// TIA Portal V17 export
// export: Created 2022-06-27T14:00:09.5735646Z, ExportSetting WithDefaults, DisplayName Totally Integrated Automation Portal, DisplayVersion V17 Update 3, DisplayName TIA Portal Openness, DisplayVersion V17 Update 3, DisplayName TIA Portal Version Control Interface, DisplayVersion V17, DisplayName SINAMICS Startdrive Advanced, DisplayVersion V17 Update1, DisplayName SINAMICS Startdrive G110M, G120, G120C, G120D, G120P, G115D, DisplayVersion V17 Update1, DisplayName SINAMICS Startdrive G130, G150, S120, S150, SINAMICS MV, S210, DisplayVersion V17 Update1, DisplayName STEP 7 Professional, DisplayVersion V17 Update 3, DisplayName STEP 7 Safety, DisplayVersion V17, DisplayName WinCC UA Professional, DisplayVersion V17 Update 3
FUNCTION_BLOCK "S0822_RECIPE_FAILURES"   // FB822, LAD
{ S7_Optimized_Access := 'TRUE' }
VERSION : 0.1
// stored: AutoNumber false, IsIECCheckEnabled false, IsRetainMemResEnabled false, MemoryReserve 100, SetENOAutomatically false, UDAEnableTagReadback false
   VAR
      ls_wFaultRecipe : Word;
      ls_dwC1FaultProfile : DWord;
      ls_dwC2FaultProfile : DWord;
      ls_bRecipeOk : Bool;
   END_VAR
BEGIN

REGION Network 1: Falha Receita - Nome Receita
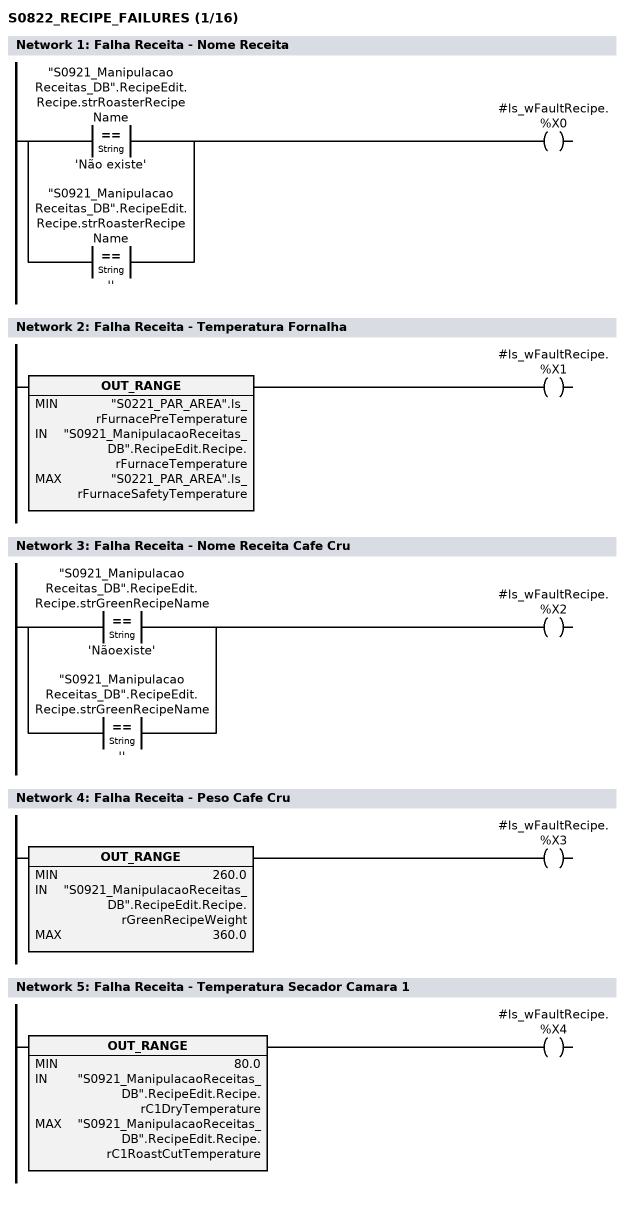
   RUNG wire#powerrail
      { S7_Templates := "SrcType := String" } EQ_Contact(in1 := "S0921_ManipulacaoReceitas_DB".RecipeEdit.Recipe.strRoasterRecipeName, in2 := 'Não existe')
      wire#w1
      Coil( #ls_wFaultRecipe.%X0 )
   END_RUNG
   RUNG wire#powerrail
      { S7_Templates := "SrcType := String" } EQ_Contact(in1 := "S0921_ManipulacaoReceitas_DB".RecipeEdit.Recipe.strRoasterRecipeName, in2 := '')
   END_RUNG wire#w1
   // the same network as SCL:
   #ls_wFaultRecipe.%X0 := ("S0921_ManipulacaoReceitas_DB".RecipeEdit.Recipe.strRoasterRecipeName = 'Não existe') OR ("S0921_ManipulacaoReceitas_DB".RecipeEdit.Recipe.strRoasterRecipeName = '');
END_REGION

REGION Network 2: Falha Receita - Temperatura Fornalha
   #ls_wFaultRecipe.%X1 := ("S0921_ManipulacaoReceitas_DB".RecipeEdit.Recipe.rFurnaceTemperature < "S0221_PAR_AREA".ls_rFurnacePreTemperature) OR ("S0921_ManipulacaoReceitas_DB".RecipeEdit.Recipe.rFurnaceTemperature > "S0221_PAR_AREA".ls_rFurnaceSafetyTemperature);
END_REGION

REGION Network 3: Falha Receita - Nome Receita Cafe Cru
   RUNG wire#powerrail
      { S7_Templates := "SrcType := String" } EQ_Contact(in1 := "S0921_ManipulacaoReceitas_DB".RecipeEdit.Recipe.strGreenRecipeName, in2 := 'Nãoexiste')
      wire#w1
      Coil( #ls_wFaultRecipe.%X2 )
   END_RUNG
   RUNG wire#powerrail
      { S7_Templates := "SrcType := String" } EQ_Contact(in1 := "S0921_ManipulacaoReceitas_DB".RecipeEdit.Recipe.strGreenRecipeName, in2 := '')
   END_RUNG wire#w1
   // the same network as SCL:
   #ls_wFaultRecipe.%X2 := ("S0921_ManipulacaoReceitas_DB".RecipeEdit.Recipe.strGreenRecipeName = 'Nãoexiste') OR ("S0921_ManipulacaoReceitas_DB".RecipeEdit.Recipe.strGreenRecipeName = '');
END_REGION

REGION Network 4: Falha Receita - Peso Cafe Cru
   #ls_wFaultRecipe.%X3 := ("S0921_ManipulacaoReceitas_DB".RecipeEdit.Recipe.rGreenRecipeWeight < 260.0) OR ("S0921_ManipulacaoReceitas_DB".RecipeEdit.Recipe.rGreenRecipeWeight > 360.0);
END_REGION

REGION Network 5: Falha Receita - Temperatura Secador Camara 1
   #ls_wFaultRecipe.%X4 := ("S0921_ManipulacaoReceitas_DB".RecipeEdit.Recipe.rC1DryTemperature < 80.0) OR ("S0921_ManipulacaoReceitas_DB".RecipeEdit.Recipe.rC1DryTemperature > "S0921_ManipulacaoReceitas_DB".RecipeEdit.Recipe.rC1RoastCutTemperature);
END_REGION

REGION Network 6: Falha Receita - Temperatura Secador Camara 2
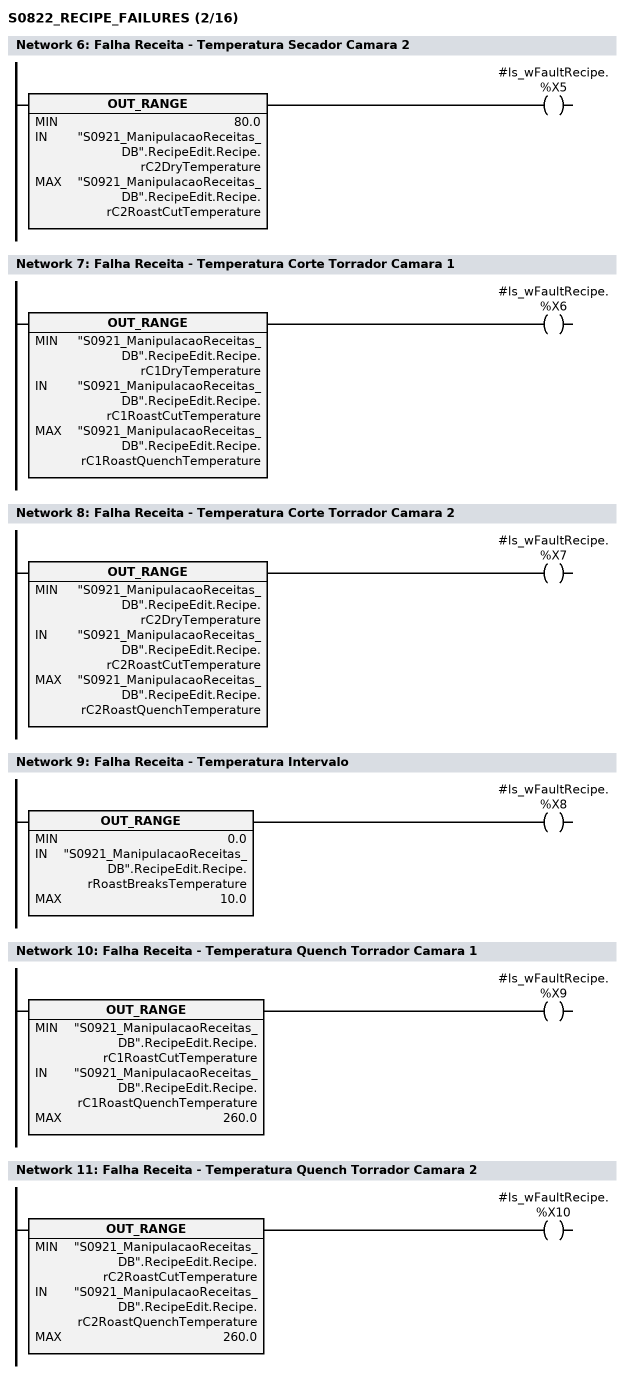
   #ls_wFaultRecipe.%X5 := ("S0921_ManipulacaoReceitas_DB".RecipeEdit.Recipe.rC2DryTemperature < 80.0) OR ("S0921_ManipulacaoReceitas_DB".RecipeEdit.Recipe.rC2DryTemperature > "S0921_ManipulacaoReceitas_DB".RecipeEdit.Recipe.rC2RoastCutTemperature);
END_REGION

REGION Network 7: Falha Receita - Temperatura Corte Torrador Camara 1
   #ls_wFaultRecipe.%X6 := ("S0921_ManipulacaoReceitas_DB".RecipeEdit.Recipe.rC1RoastCutTemperature < "S0921_ManipulacaoReceitas_DB".RecipeEdit.Recipe.rC1DryTemperature) OR ("S0921_ManipulacaoReceitas_DB".RecipeEdit.Recipe.rC1RoastCutTemperature > "S0921_ManipulacaoReceitas_DB".RecipeEdit.Recipe.rC1RoastQuenchTemperature);
END_REGION

REGION Network 8: Falha Receita - Temperatura Corte Torrador Camara 2
   #ls_wFaultRecipe.%X7 := ("S0921_ManipulacaoReceitas_DB".RecipeEdit.Recipe.rC2RoastCutTemperature < "S0921_ManipulacaoReceitas_DB".RecipeEdit.Recipe.rC2DryTemperature) OR ("S0921_ManipulacaoReceitas_DB".RecipeEdit.Recipe.rC2RoastCutTemperature > "S0921_ManipulacaoReceitas_DB".RecipeEdit.Recipe.rC2RoastQuenchTemperature);
END_REGION

REGION Network 9: Falha Receita - Temperatura Intervalo
   #ls_wFaultRecipe.%X8 := ("S0921_ManipulacaoReceitas_DB".RecipeEdit.Recipe.rRoastBreaksTemperature < 0.0) OR ("S0921_ManipulacaoReceitas_DB".RecipeEdit.Recipe.rRoastBreaksTemperature > 10.0);
END_REGION

REGION Network 10: Falha Receita - Temperatura Quench Torrador Camara 1
   #ls_wFaultRecipe.%X9 := ("S0921_ManipulacaoReceitas_DB".RecipeEdit.Recipe.rC1RoastQuenchTemperature < "S0921_ManipulacaoReceitas_DB".RecipeEdit.Recipe.rC1RoastCutTemperature) OR ("S0921_ManipulacaoReceitas_DB".RecipeEdit.Recipe.rC1RoastQuenchTemperature > 260.0);
END_REGION

REGION Network 11: Falha Receita - Temperatura Quench Torrador Camara 2
   #ls_wFaultRecipe.%X10 := ("S0921_ManipulacaoReceitas_DB".RecipeEdit.Recipe.rC2RoastQuenchTemperature < "S0921_ManipulacaoReceitas_DB".RecipeEdit.Recipe.rC2RoastCutTemperature) OR ("S0921_ManipulacaoReceitas_DB".RecipeEdit.Recipe.rC2RoastQuenchTemperature > 260.0);
END_REGION

REGION Network 12: Falha Receita - Total Quench Torrador Camara 1
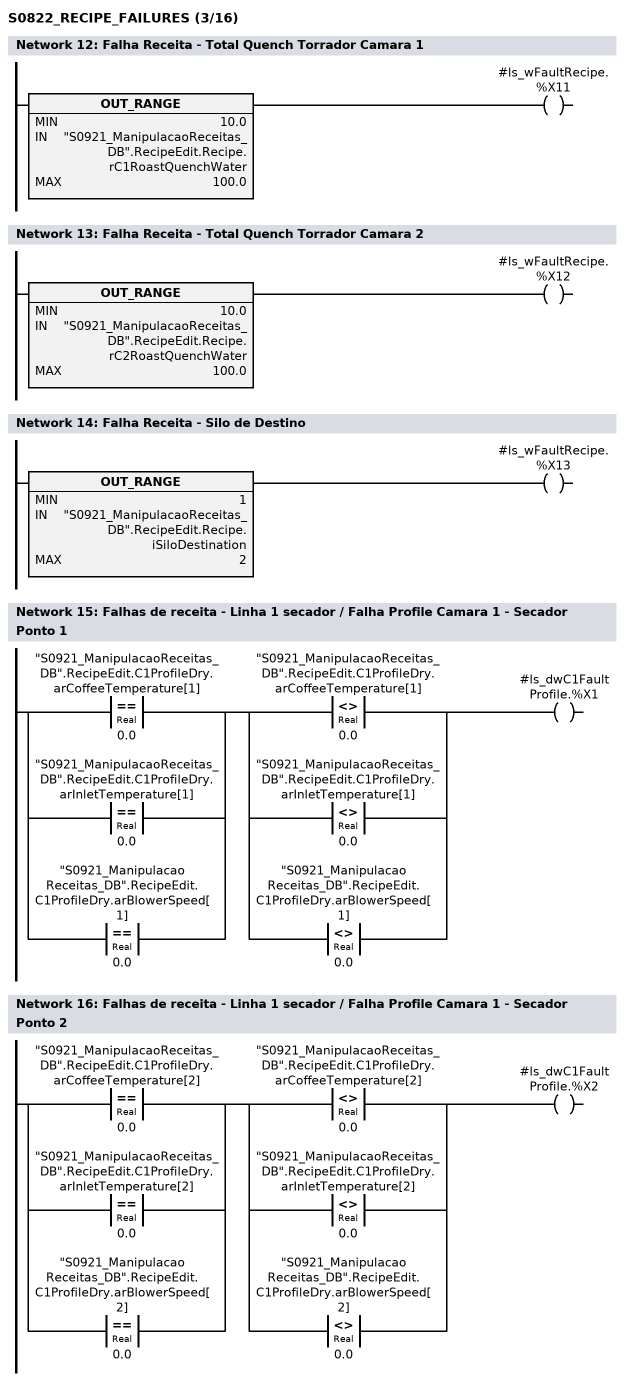
   #ls_wFaultRecipe.%X11 := ("S0921_ManipulacaoReceitas_DB".RecipeEdit.Recipe.rC1RoastQuenchWater < 10.0) OR ("S0921_ManipulacaoReceitas_DB".RecipeEdit.Recipe.rC1RoastQuenchWater > 100.0);
END_REGION

REGION Network 13: Falha Receita - Total Quench Torrador Camara 2
   #ls_wFaultRecipe.%X12 := ("S0921_ManipulacaoReceitas_DB".RecipeEdit.Recipe.rC2RoastQuenchWater < 10.0) OR ("S0921_ManipulacaoReceitas_DB".RecipeEdit.Recipe.rC2RoastQuenchWater > 100.0);
END_REGION

REGION Network 14: Falha Receita - Silo de Destino
   #ls_wFaultRecipe.%X13 := ("S0921_ManipulacaoReceitas_DB".RecipeEdit.Recipe.iSiloDestination < 1) OR ("S0921_ManipulacaoReceitas_DB".RecipeEdit.Recipe.iSiloDestination > 2);
END_REGION

REGION Network 15: Falhas de receita - Linha 1 secador / Falha Profile Camara 1 - Secador Ponto 1
   RUNG wire#powerrail
      { S7_Templates := "SrcType := Real" } EQ_Contact(in1 := "S0921_ManipulacaoReceitas_DB".RecipeEdit.C1ProfileDry.arCoffeeTemperature[1], in2 := 0.0)
      wire#w1
      { S7_Templates := "SrcType := Real" } NE_Contact(in1 := "S0921_ManipulacaoReceitas_DB".RecipeEdit.C1ProfileDry.arCoffeeTemperature[1], in2 := 0.0)
      wire#w2
      Coil( #ls_dwC1FaultProfile.%X1 )
   END_RUNG
   RUNG wire#powerrail
      { S7_Templates := "SrcType := Real" } EQ_Contact(in1 := "S0921_ManipulacaoReceitas_DB".RecipeEdit.C1ProfileDry.arInletTemperature[1], in2 := 0.0)
   END_RUNG wire#w1
   RUNG wire#powerrail
      { S7_Templates := "SrcType := Real" } EQ_Contact(in1 := "S0921_ManipulacaoReceitas_DB".RecipeEdit.C1ProfileDry.arBlowerSpeed[1], in2 := 0.0)
   END_RUNG wire#w1
   RUNG wire#w1
      { S7_Templates := "SrcType := Real" } NE_Contact(in1 := "S0921_ManipulacaoReceitas_DB".RecipeEdit.C1ProfileDry.arInletTemperature[1], in2 := 0.0)
   END_RUNG wire#w2
   RUNG wire#w1
      { S7_Templates := "SrcType := Real" } NE_Contact(in1 := "S0921_ManipulacaoReceitas_DB".RecipeEdit.C1ProfileDry.arBlowerSpeed[1], in2 := 0.0)
   END_RUNG wire#w2
   // the same network as SCL:
   #ls_dwC1FaultProfile.%X1 := (("S0921_ManipulacaoReceitas_DB".RecipeEdit.C1ProfileDry.arCoffeeTemperature[1] = 0.0) OR ("S0921_ManipulacaoReceitas_DB".RecipeEdit.C1ProfileDry.arInletTemperature[1] = 0.0) OR ("S0921_ManipulacaoReceitas_DB".RecipeEdit.C1ProfileDry.arBlowerSpeed[1] = 0.0)) AND (("S0921_ManipulacaoReceitas_DB".RecipeEdit.C1ProfileDry.arCoffeeTemperature[1] <> 0.0) OR ("S0921_ManipulacaoReceitas_DB".RecipeEdit.C1ProfileDry.arInletTemperature[1] <> 0.0) OR ("S0921_ManipulacaoReceitas_DB".RecipeEdit.C1ProfileDry.arBlowerSpeed[1] <> 0.0));
END_REGION

REGION Network 16: Falhas de receita - Linha 1 secador / Falha Profile Camara 1 - Secador Ponto 2
   RUNG wire#powerrail
      { S7_Templates := "SrcType := Real" } EQ_Contact(in1 := "S0921_ManipulacaoReceitas_DB".RecipeEdit.C1ProfileDry.arCoffeeTemperature[2], in2 := 0.0)
      wire#w1
      { S7_Templates := "SrcType := Real" } NE_Contact(in1 := "S0921_ManipulacaoReceitas_DB".RecipeEdit.C1ProfileDry.arCoffeeTemperature[2], in2 := 0.0)
      wire#w2
      Coil( #ls_dwC1FaultProfile.%X2 )
   END_RUNG
   RUNG wire#powerrail
      { S7_Templates := "SrcType := Real" } EQ_Contact(in1 := "S0921_ManipulacaoReceitas_DB".RecipeEdit.C1ProfileDry.arInletTemperature[2], in2 := 0.0)
   END_RUNG wire#w1
   RUNG wire#powerrail
      { S7_Templates := "SrcType := Real" } EQ_Contact(in1 := "S0921_ManipulacaoReceitas_DB".RecipeEdit.C1ProfileDry.arBlowerSpeed[2], in2 := 0.0)
   END_RUNG wire#w1
   RUNG wire#w1
      { S7_Templates := "SrcType := Real" } NE_Contact(in1 := "S0921_ManipulacaoReceitas_DB".RecipeEdit.C1ProfileDry.arInletTemperature[2], in2 := 0.0)
   END_RUNG wire#w2
   RUNG wire#w1
      { S7_Templates := "SrcType := Real" } NE_Contact(in1 := "S0921_ManipulacaoReceitas_DB".RecipeEdit.C1ProfileDry.arBlowerSpeed[2], in2 := 0.0)
   END_RUNG wire#w2
   // the same network as SCL:
   #ls_dwC1FaultProfile.%X2 := (("S0921_ManipulacaoReceitas_DB".RecipeEdit.C1ProfileDry.arCoffeeTemperature[2] = 0.0) OR ("S0921_ManipulacaoReceitas_DB".RecipeEdit.C1ProfileDry.arInletTemperature[2] = 0.0) OR ("S0921_ManipulacaoReceitas_DB".RecipeEdit.C1ProfileDry.arBlowerSpeed[2] = 0.0)) AND (("S0921_ManipulacaoReceitas_DB".RecipeEdit.C1ProfileDry.arCoffeeTemperature[2] <> 0.0) OR ("S0921_ManipulacaoReceitas_DB".RecipeEdit.C1ProfileDry.arInletTemperature[2] <> 0.0) OR ("S0921_ManipulacaoReceitas_DB".RecipeEdit.C1ProfileDry.arBlowerSpeed[2] <> 0.0));
END_REGION

REGION Network 17: Falhas de receita - Linha 1 secador / Falha Profile Camara 1 - Secador Ponto 3
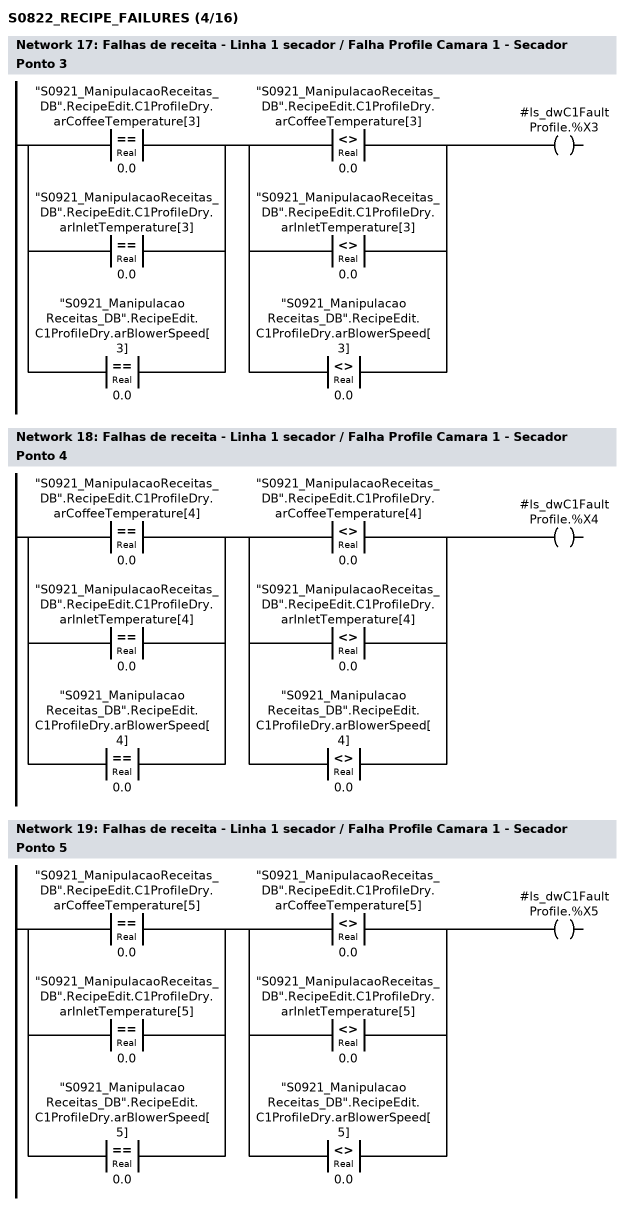
   RUNG wire#powerrail
      { S7_Templates := "SrcType := Real" } EQ_Contact(in1 := "S0921_ManipulacaoReceitas_DB".RecipeEdit.C1ProfileDry.arCoffeeTemperature[3], in2 := 0.0)
      wire#w1
      { S7_Templates := "SrcType := Real" } NE_Contact(in1 := "S0921_ManipulacaoReceitas_DB".RecipeEdit.C1ProfileDry.arCoffeeTemperature[3], in2 := 0.0)
      wire#w2
      Coil( #ls_dwC1FaultProfile.%X3 )
   END_RUNG
   RUNG wire#powerrail
      { S7_Templates := "SrcType := Real" } EQ_Contact(in1 := "S0921_ManipulacaoReceitas_DB".RecipeEdit.C1ProfileDry.arInletTemperature[3], in2 := 0.0)
   END_RUNG wire#w1
   RUNG wire#powerrail
      { S7_Templates := "SrcType := Real" } EQ_Contact(in1 := "S0921_ManipulacaoReceitas_DB".RecipeEdit.C1ProfileDry.arBlowerSpeed[3], in2 := 0.0)
   END_RUNG wire#w1
   RUNG wire#w1
      { S7_Templates := "SrcType := Real" } NE_Contact(in1 := "S0921_ManipulacaoReceitas_DB".RecipeEdit.C1ProfileDry.arInletTemperature[3], in2 := 0.0)
   END_RUNG wire#w2
   RUNG wire#w1
      { S7_Templates := "SrcType := Real" } NE_Contact(in1 := "S0921_ManipulacaoReceitas_DB".RecipeEdit.C1ProfileDry.arBlowerSpeed[3], in2 := 0.0)
   END_RUNG wire#w2
   // the same network as SCL:
   #ls_dwC1FaultProfile.%X3 := (("S0921_ManipulacaoReceitas_DB".RecipeEdit.C1ProfileDry.arCoffeeTemperature[3] = 0.0) OR ("S0921_ManipulacaoReceitas_DB".RecipeEdit.C1ProfileDry.arInletTemperature[3] = 0.0) OR ("S0921_ManipulacaoReceitas_DB".RecipeEdit.C1ProfileDry.arBlowerSpeed[3] = 0.0)) AND (("S0921_ManipulacaoReceitas_DB".RecipeEdit.C1ProfileDry.arCoffeeTemperature[3] <> 0.0) OR ("S0921_ManipulacaoReceitas_DB".RecipeEdit.C1ProfileDry.arInletTemperature[3] <> 0.0) OR ("S0921_ManipulacaoReceitas_DB".RecipeEdit.C1ProfileDry.arBlowerSpeed[3] <> 0.0));
END_REGION

REGION Network 18: Falhas de receita - Linha 1 secador / Falha Profile Camara 1 - Secador Ponto 4
   RUNG wire#powerrail
      { S7_Templates := "SrcType := Real" } EQ_Contact(in1 := "S0921_ManipulacaoReceitas_DB".RecipeEdit.C1ProfileDry.arCoffeeTemperature[4], in2 := 0.0)
      wire#w1
      { S7_Templates := "SrcType := Real" } NE_Contact(in1 := "S0921_ManipulacaoReceitas_DB".RecipeEdit.C1ProfileDry.arCoffeeTemperature[4], in2 := 0.0)
      wire#w2
      Coil( #ls_dwC1FaultProfile.%X4 )
   END_RUNG
   RUNG wire#powerrail
      { S7_Templates := "SrcType := Real" } EQ_Contact(in1 := "S0921_ManipulacaoReceitas_DB".RecipeEdit.C1ProfileDry.arInletTemperature[4], in2 := 0.0)
   END_RUNG wire#w1
   RUNG wire#powerrail
      { S7_Templates := "SrcType := Real" } EQ_Contact(in1 := "S0921_ManipulacaoReceitas_DB".RecipeEdit.C1ProfileDry.arBlowerSpeed[4], in2 := 0.0)
   END_RUNG wire#w1
   RUNG wire#w1
      { S7_Templates := "SrcType := Real" } NE_Contact(in1 := "S0921_ManipulacaoReceitas_DB".RecipeEdit.C1ProfileDry.arInletTemperature[4], in2 := 0.0)
   END_RUNG wire#w2
   RUNG wire#w1
      { S7_Templates := "SrcType := Real" } NE_Contact(in1 := "S0921_ManipulacaoReceitas_DB".RecipeEdit.C1ProfileDry.arBlowerSpeed[4], in2 := 0.0)
   END_RUNG wire#w2
   // the same network as SCL:
   #ls_dwC1FaultProfile.%X4 := (("S0921_ManipulacaoReceitas_DB".RecipeEdit.C1ProfileDry.arCoffeeTemperature[4] = 0.0) OR ("S0921_ManipulacaoReceitas_DB".RecipeEdit.C1ProfileDry.arInletTemperature[4] = 0.0) OR ("S0921_ManipulacaoReceitas_DB".RecipeEdit.C1ProfileDry.arBlowerSpeed[4] = 0.0)) AND (("S0921_ManipulacaoReceitas_DB".RecipeEdit.C1ProfileDry.arCoffeeTemperature[4] <> 0.0) OR ("S0921_ManipulacaoReceitas_DB".RecipeEdit.C1ProfileDry.arInletTemperature[4] <> 0.0) OR ("S0921_ManipulacaoReceitas_DB".RecipeEdit.C1ProfileDry.arBlowerSpeed[4] <> 0.0));
END_REGION

REGION Network 19: Falhas de receita - Linha 1 secador / Falha Profile Camara 1 - Secador Ponto 5
   RUNG wire#powerrail
      { S7_Templates := "SrcType := Real" } EQ_Contact(in1 := "S0921_ManipulacaoReceitas_DB".RecipeEdit.C1ProfileDry.arCoffeeTemperature[5], in2 := 0.0)
      wire#w1
      { S7_Templates := "SrcType := Real" } NE_Contact(in1 := "S0921_ManipulacaoReceitas_DB".RecipeEdit.C1ProfileDry.arCoffeeTemperature[5], in2 := 0.0)
      wire#w2
      Coil( #ls_dwC1FaultProfile.%X5 )
   END_RUNG
   RUNG wire#powerrail
      { S7_Templates := "SrcType := Real" } EQ_Contact(in1 := "S0921_ManipulacaoReceitas_DB".RecipeEdit.C1ProfileDry.arInletTemperature[5], in2 := 0.0)
   END_RUNG wire#w1
   RUNG wire#powerrail
      { S7_Templates := "SrcType := Real" } EQ_Contact(in1 := "S0921_ManipulacaoReceitas_DB".RecipeEdit.C1ProfileDry.arBlowerSpeed[5], in2 := 0.0)
   END_RUNG wire#w1
   RUNG wire#w1
      { S7_Templates := "SrcType := Real" } NE_Contact(in1 := "S0921_ManipulacaoReceitas_DB".RecipeEdit.C1ProfileDry.arInletTemperature[5], in2 := 0.0)
   END_RUNG wire#w2
   RUNG wire#w1
      { S7_Templates := "SrcType := Real" } NE_Contact(in1 := "S0921_ManipulacaoReceitas_DB".RecipeEdit.C1ProfileDry.arBlowerSpeed[5], in2 := 0.0)
   END_RUNG wire#w2
   // the same network as SCL:
   #ls_dwC1FaultProfile.%X5 := (("S0921_ManipulacaoReceitas_DB".RecipeEdit.C1ProfileDry.arCoffeeTemperature[5] = 0.0) OR ("S0921_ManipulacaoReceitas_DB".RecipeEdit.C1ProfileDry.arInletTemperature[5] = 0.0) OR ("S0921_ManipulacaoReceitas_DB".RecipeEdit.C1ProfileDry.arBlowerSpeed[5] = 0.0)) AND (("S0921_ManipulacaoReceitas_DB".RecipeEdit.C1ProfileDry.arCoffeeTemperature[5] <> 0.0) OR ("S0921_ManipulacaoReceitas_DB".RecipeEdit.C1ProfileDry.arInletTemperature[5] <> 0.0) OR ("S0921_ManipulacaoReceitas_DB".RecipeEdit.C1ProfileDry.arBlowerSpeed[5] <> 0.0));
END_REGION

REGION Network 20: Falhas de receita - Linha 1 secador / Falha Profile Camara 1 - Secador Ponto 6
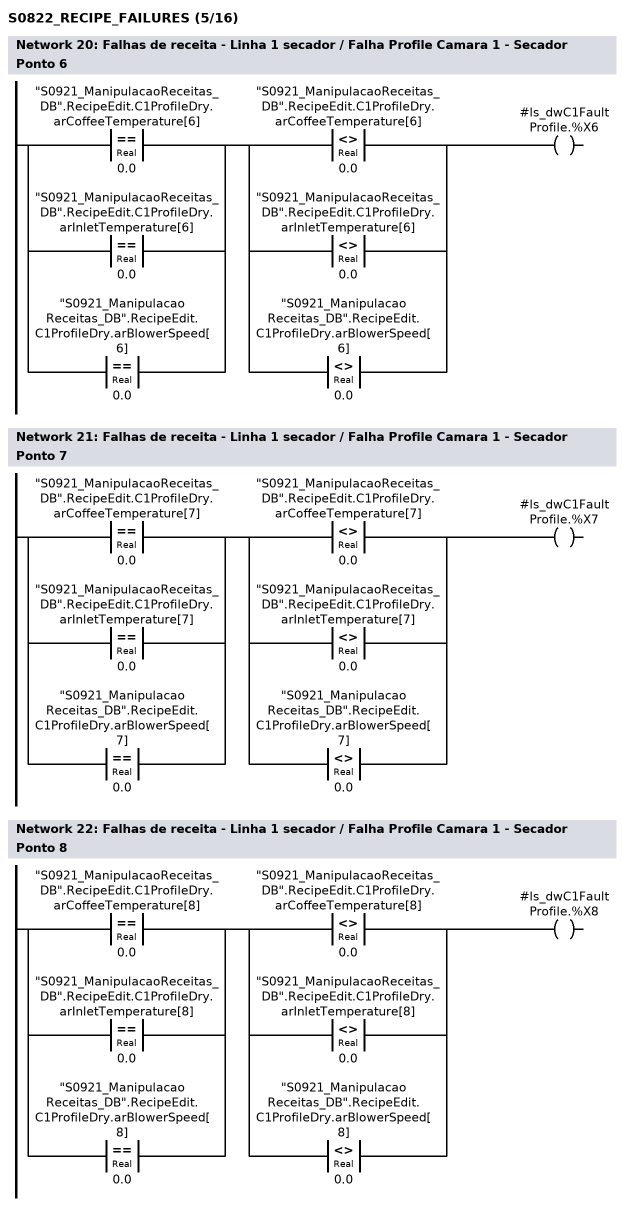
   RUNG wire#powerrail
      { S7_Templates := "SrcType := Real" } EQ_Contact(in1 := "S0921_ManipulacaoReceitas_DB".RecipeEdit.C1ProfileDry.arCoffeeTemperature[6], in2 := 0.0)
      wire#w1
      { S7_Templates := "SrcType := Real" } NE_Contact(in1 := "S0921_ManipulacaoReceitas_DB".RecipeEdit.C1ProfileDry.arCoffeeTemperature[6], in2 := 0.0)
      wire#w2
      Coil( #ls_dwC1FaultProfile.%X6 )
   END_RUNG
   RUNG wire#powerrail
      { S7_Templates := "SrcType := Real" } EQ_Contact(in1 := "S0921_ManipulacaoReceitas_DB".RecipeEdit.C1ProfileDry.arInletTemperature[6], in2 := 0.0)
   END_RUNG wire#w1
   RUNG wire#powerrail
      { S7_Templates := "SrcType := Real" } EQ_Contact(in1 := "S0921_ManipulacaoReceitas_DB".RecipeEdit.C1ProfileDry.arBlowerSpeed[6], in2 := 0.0)
   END_RUNG wire#w1
   RUNG wire#w1
      { S7_Templates := "SrcType := Real" } NE_Contact(in1 := "S0921_ManipulacaoReceitas_DB".RecipeEdit.C1ProfileDry.arInletTemperature[6], in2 := 0.0)
   END_RUNG wire#w2
   RUNG wire#w1
      { S7_Templates := "SrcType := Real" } NE_Contact(in1 := "S0921_ManipulacaoReceitas_DB".RecipeEdit.C1ProfileDry.arBlowerSpeed[6], in2 := 0.0)
   END_RUNG wire#w2
   // the same network as SCL:
   #ls_dwC1FaultProfile.%X6 := (("S0921_ManipulacaoReceitas_DB".RecipeEdit.C1ProfileDry.arCoffeeTemperature[6] = 0.0) OR ("S0921_ManipulacaoReceitas_DB".RecipeEdit.C1ProfileDry.arInletTemperature[6] = 0.0) OR ("S0921_ManipulacaoReceitas_DB".RecipeEdit.C1ProfileDry.arBlowerSpeed[6] = 0.0)) AND (("S0921_ManipulacaoReceitas_DB".RecipeEdit.C1ProfileDry.arCoffeeTemperature[6] <> 0.0) OR ("S0921_ManipulacaoReceitas_DB".RecipeEdit.C1ProfileDry.arInletTemperature[6] <> 0.0) OR ("S0921_ManipulacaoReceitas_DB".RecipeEdit.C1ProfileDry.arBlowerSpeed[6] <> 0.0));
END_REGION

REGION Network 21: Falhas de receita - Linha 1 secador / Falha Profile Camara 1 - Secador Ponto 7
   RUNG wire#powerrail
      { S7_Templates := "SrcType := Real" } EQ_Contact(in1 := "S0921_ManipulacaoReceitas_DB".RecipeEdit.C1ProfileDry.arCoffeeTemperature[7], in2 := 0.0)
      wire#w1
      { S7_Templates := "SrcType := Real" } NE_Contact(in1 := "S0921_ManipulacaoReceitas_DB".RecipeEdit.C1ProfileDry.arCoffeeTemperature[7], in2 := 0.0)
      wire#w2
      Coil( #ls_dwC1FaultProfile.%X7 )
   END_RUNG
   RUNG wire#powerrail
      { S7_Templates := "SrcType := Real" } EQ_Contact(in1 := "S0921_ManipulacaoReceitas_DB".RecipeEdit.C1ProfileDry.arInletTemperature[7], in2 := 0.0)
   END_RUNG wire#w1
   RUNG wire#powerrail
      { S7_Templates := "SrcType := Real" } EQ_Contact(in1 := "S0921_ManipulacaoReceitas_DB".RecipeEdit.C1ProfileDry.arBlowerSpeed[7], in2 := 0.0)
   END_RUNG wire#w1
   RUNG wire#w1
      { S7_Templates := "SrcType := Real" } NE_Contact(in1 := "S0921_ManipulacaoReceitas_DB".RecipeEdit.C1ProfileDry.arInletTemperature[7], in2 := 0.0)
   END_RUNG wire#w2
   RUNG wire#w1
      { S7_Templates := "SrcType := Real" } NE_Contact(in1 := "S0921_ManipulacaoReceitas_DB".RecipeEdit.C1ProfileDry.arBlowerSpeed[7], in2 := 0.0)
   END_RUNG wire#w2
   // the same network as SCL:
   #ls_dwC1FaultProfile.%X7 := (("S0921_ManipulacaoReceitas_DB".RecipeEdit.C1ProfileDry.arCoffeeTemperature[7] = 0.0) OR ("S0921_ManipulacaoReceitas_DB".RecipeEdit.C1ProfileDry.arInletTemperature[7] = 0.0) OR ("S0921_ManipulacaoReceitas_DB".RecipeEdit.C1ProfileDry.arBlowerSpeed[7] = 0.0)) AND (("S0921_ManipulacaoReceitas_DB".RecipeEdit.C1ProfileDry.arCoffeeTemperature[7] <> 0.0) OR ("S0921_ManipulacaoReceitas_DB".RecipeEdit.C1ProfileDry.arInletTemperature[7] <> 0.0) OR ("S0921_ManipulacaoReceitas_DB".RecipeEdit.C1ProfileDry.arBlowerSpeed[7] <> 0.0));
END_REGION

REGION Network 22: Falhas de receita - Linha 1 secador / Falha Profile Camara 1 - Secador Ponto 8
   RUNG wire#powerrail
      { S7_Templates := "SrcType := Real" } EQ_Contact(in1 := "S0921_ManipulacaoReceitas_DB".RecipeEdit.C1ProfileDry.arCoffeeTemperature[8], in2 := 0.0)
      wire#w1
      { S7_Templates := "SrcType := Real" } NE_Contact(in1 := "S0921_ManipulacaoReceitas_DB".RecipeEdit.C1ProfileDry.arCoffeeTemperature[8], in2 := 0.0)
      wire#w2
      Coil( #ls_dwC1FaultProfile.%X8 )
   END_RUNG
   RUNG wire#powerrail
      { S7_Templates := "SrcType := Real" } EQ_Contact(in1 := "S0921_ManipulacaoReceitas_DB".RecipeEdit.C1ProfileDry.arInletTemperature[8], in2 := 0.0)
   END_RUNG wire#w1
   RUNG wire#powerrail
      { S7_Templates := "SrcType := Real" } EQ_Contact(in1 := "S0921_ManipulacaoReceitas_DB".RecipeEdit.C1ProfileDry.arBlowerSpeed[8], in2 := 0.0)
   END_RUNG wire#w1
   RUNG wire#w1
      { S7_Templates := "SrcType := Real" } NE_Contact(in1 := "S0921_ManipulacaoReceitas_DB".RecipeEdit.C1ProfileDry.arInletTemperature[8], in2 := 0.0)
   END_RUNG wire#w2
   RUNG wire#w1
      { S7_Templates := "SrcType := Real" } NE_Contact(in1 := "S0921_ManipulacaoReceitas_DB".RecipeEdit.C1ProfileDry.arBlowerSpeed[8], in2 := 0.0)
   END_RUNG wire#w2
   // the same network as SCL:
   #ls_dwC1FaultProfile.%X8 := (("S0921_ManipulacaoReceitas_DB".RecipeEdit.C1ProfileDry.arCoffeeTemperature[8] = 0.0) OR ("S0921_ManipulacaoReceitas_DB".RecipeEdit.C1ProfileDry.arInletTemperature[8] = 0.0) OR ("S0921_ManipulacaoReceitas_DB".RecipeEdit.C1ProfileDry.arBlowerSpeed[8] = 0.0)) AND (("S0921_ManipulacaoReceitas_DB".RecipeEdit.C1ProfileDry.arCoffeeTemperature[8] <> 0.0) OR ("S0921_ManipulacaoReceitas_DB".RecipeEdit.C1ProfileDry.arInletTemperature[8] <> 0.0) OR ("S0921_ManipulacaoReceitas_DB".RecipeEdit.C1ProfileDry.arBlowerSpeed[8] <> 0.0));
END_REGION

REGION Network 23: Falhas de receita - Linha 1 secador / Falha Profile Camara 1 - Secador Ponto 9
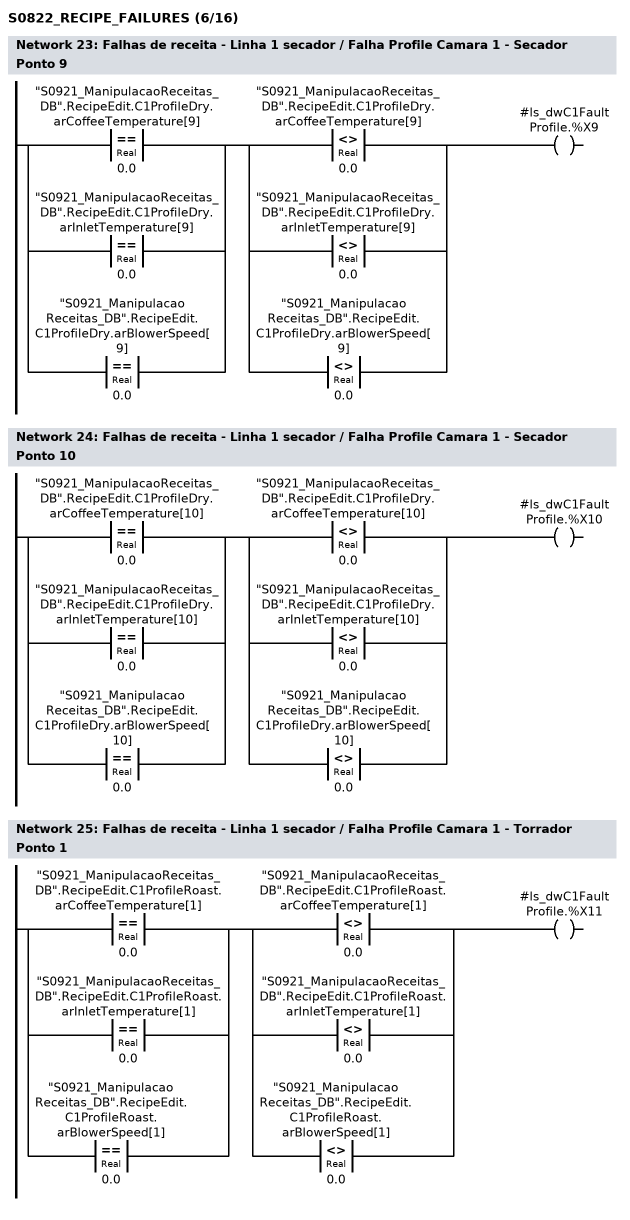
   RUNG wire#powerrail
      { S7_Templates := "SrcType := Real" } EQ_Contact(in1 := "S0921_ManipulacaoReceitas_DB".RecipeEdit.C1ProfileDry.arCoffeeTemperature[9], in2 := 0.0)
      wire#w1
      { S7_Templates := "SrcType := Real" } NE_Contact(in1 := "S0921_ManipulacaoReceitas_DB".RecipeEdit.C1ProfileDry.arCoffeeTemperature[9], in2 := 0.0)
      wire#w2
      Coil( #ls_dwC1FaultProfile.%X9 )
   END_RUNG
   RUNG wire#powerrail
      { S7_Templates := "SrcType := Real" } EQ_Contact(in1 := "S0921_ManipulacaoReceitas_DB".RecipeEdit.C1ProfileDry.arInletTemperature[9], in2 := 0.0)
   END_RUNG wire#w1
   RUNG wire#powerrail
      { S7_Templates := "SrcType := Real" } EQ_Contact(in1 := "S0921_ManipulacaoReceitas_DB".RecipeEdit.C1ProfileDry.arBlowerSpeed[9], in2 := 0.0)
   END_RUNG wire#w1
   RUNG wire#w1
      { S7_Templates := "SrcType := Real" } NE_Contact(in1 := "S0921_ManipulacaoReceitas_DB".RecipeEdit.C1ProfileDry.arInletTemperature[9], in2 := 0.0)
   END_RUNG wire#w2
   RUNG wire#w1
      { S7_Templates := "SrcType := Real" } NE_Contact(in1 := "S0921_ManipulacaoReceitas_DB".RecipeEdit.C1ProfileDry.arBlowerSpeed[9], in2 := 0.0)
   END_RUNG wire#w2
   // the same network as SCL:
   #ls_dwC1FaultProfile.%X9 := (("S0921_ManipulacaoReceitas_DB".RecipeEdit.C1ProfileDry.arCoffeeTemperature[9] = 0.0) OR ("S0921_ManipulacaoReceitas_DB".RecipeEdit.C1ProfileDry.arInletTemperature[9] = 0.0) OR ("S0921_ManipulacaoReceitas_DB".RecipeEdit.C1ProfileDry.arBlowerSpeed[9] = 0.0)) AND (("S0921_ManipulacaoReceitas_DB".RecipeEdit.C1ProfileDry.arCoffeeTemperature[9] <> 0.0) OR ("S0921_ManipulacaoReceitas_DB".RecipeEdit.C1ProfileDry.arInletTemperature[9] <> 0.0) OR ("S0921_ManipulacaoReceitas_DB".RecipeEdit.C1ProfileDry.arBlowerSpeed[9] <> 0.0));
END_REGION

REGION Network 24: Falhas de receita - Linha 1 secador / Falha Profile Camara 1 - Secador Ponto 10
   RUNG wire#powerrail
      { S7_Templates := "SrcType := Real" } EQ_Contact(in1 := "S0921_ManipulacaoReceitas_DB".RecipeEdit.C1ProfileDry.arCoffeeTemperature[10], in2 := 0.0)
      wire#w1
      { S7_Templates := "SrcType := Real" } NE_Contact(in1 := "S0921_ManipulacaoReceitas_DB".RecipeEdit.C1ProfileDry.arCoffeeTemperature[10], in2 := 0.0)
      wire#w2
      Coil( #ls_dwC1FaultProfile.%X10 )
   END_RUNG
   RUNG wire#powerrail
      { S7_Templates := "SrcType := Real" } EQ_Contact(in1 := "S0921_ManipulacaoReceitas_DB".RecipeEdit.C1ProfileDry.arInletTemperature[10], in2 := 0.0)
   END_RUNG wire#w1
   RUNG wire#powerrail
      { S7_Templates := "SrcType := Real" } EQ_Contact(in1 := "S0921_ManipulacaoReceitas_DB".RecipeEdit.C1ProfileDry.arBlowerSpeed[10], in2 := 0.0)
   END_RUNG wire#w1
   RUNG wire#w1
      { S7_Templates := "SrcType := Real" } NE_Contact(in1 := "S0921_ManipulacaoReceitas_DB".RecipeEdit.C1ProfileDry.arInletTemperature[10], in2 := 0.0)
   END_RUNG wire#w2
   RUNG wire#w1
      { S7_Templates := "SrcType := Real" } NE_Contact(in1 := "S0921_ManipulacaoReceitas_DB".RecipeEdit.C1ProfileDry.arBlowerSpeed[10], in2 := 0.0)
   END_RUNG wire#w2
   // the same network as SCL:
   #ls_dwC1FaultProfile.%X10 := (("S0921_ManipulacaoReceitas_DB".RecipeEdit.C1ProfileDry.arCoffeeTemperature[10] = 0.0) OR ("S0921_ManipulacaoReceitas_DB".RecipeEdit.C1ProfileDry.arInletTemperature[10] = 0.0) OR ("S0921_ManipulacaoReceitas_DB".RecipeEdit.C1ProfileDry.arBlowerSpeed[10] = 0.0)) AND (("S0921_ManipulacaoReceitas_DB".RecipeEdit.C1ProfileDry.arCoffeeTemperature[10] <> 0.0) OR ("S0921_ManipulacaoReceitas_DB".RecipeEdit.C1ProfileDry.arInletTemperature[10] <> 0.0) OR ("S0921_ManipulacaoReceitas_DB".RecipeEdit.C1ProfileDry.arBlowerSpeed[10] <> 0.0));
END_REGION

REGION Network 25: Falhas de receita - Linha 1 secador / Falha Profile Camara 1 - Torrador Ponto 1
   RUNG wire#powerrail
      { S7_Templates := "SrcType := Real" } EQ_Contact(in1 := "S0921_ManipulacaoReceitas_DB".RecipeEdit.C1ProfileRoast.arCoffeeTemperature[1], in2 := 0.0)
      wire#w1
      { S7_Templates := "SrcType := Real" } NE_Contact(in1 := "S0921_ManipulacaoReceitas_DB".RecipeEdit.C1ProfileRoast.arCoffeeTemperature[1], in2 := 0.0)
      wire#w2
      Coil( #ls_dwC1FaultProfile.%X11 )
   END_RUNG
   RUNG wire#powerrail
      { S7_Templates := "SrcType := Real" } EQ_Contact(in1 := "S0921_ManipulacaoReceitas_DB".RecipeEdit.C1ProfileRoast.arInletTemperature[1], in2 := 0.0)
   END_RUNG wire#w1
   RUNG wire#powerrail
      { S7_Templates := "SrcType := Real" } EQ_Contact(in1 := "S0921_ManipulacaoReceitas_DB".RecipeEdit.C1ProfileRoast.arBlowerSpeed[1], in2 := 0.0)
   END_RUNG wire#w1
   RUNG wire#w1
      { S7_Templates := "SrcType := Real" } NE_Contact(in1 := "S0921_ManipulacaoReceitas_DB".RecipeEdit.C1ProfileRoast.arInletTemperature[1], in2 := 0.0)
   END_RUNG wire#w2
   RUNG wire#w1
      { S7_Templates := "SrcType := Real" } NE_Contact(in1 := "S0921_ManipulacaoReceitas_DB".RecipeEdit.C1ProfileRoast.arBlowerSpeed[1], in2 := 0.0)
   END_RUNG wire#w2
   // the same network as SCL:
   #ls_dwC1FaultProfile.%X11 := (("S0921_ManipulacaoReceitas_DB".RecipeEdit.C1ProfileRoast.arCoffeeTemperature[1] = 0.0) OR ("S0921_ManipulacaoReceitas_DB".RecipeEdit.C1ProfileRoast.arInletTemperature[1] = 0.0) OR ("S0921_ManipulacaoReceitas_DB".RecipeEdit.C1ProfileRoast.arBlowerSpeed[1] = 0.0)) AND (("S0921_ManipulacaoReceitas_DB".RecipeEdit.C1ProfileRoast.arCoffeeTemperature[1] <> 0.0) OR ("S0921_ManipulacaoReceitas_DB".RecipeEdit.C1ProfileRoast.arInletTemperature[1] <> 0.0) OR ("S0921_ManipulacaoReceitas_DB".RecipeEdit.C1ProfileRoast.arBlowerSpeed[1] <> 0.0));
END_REGION

REGION Network 26: Falhas de receita - Linha 1 secador / Falha Profile Camara 1 - Torrador Ponto 2
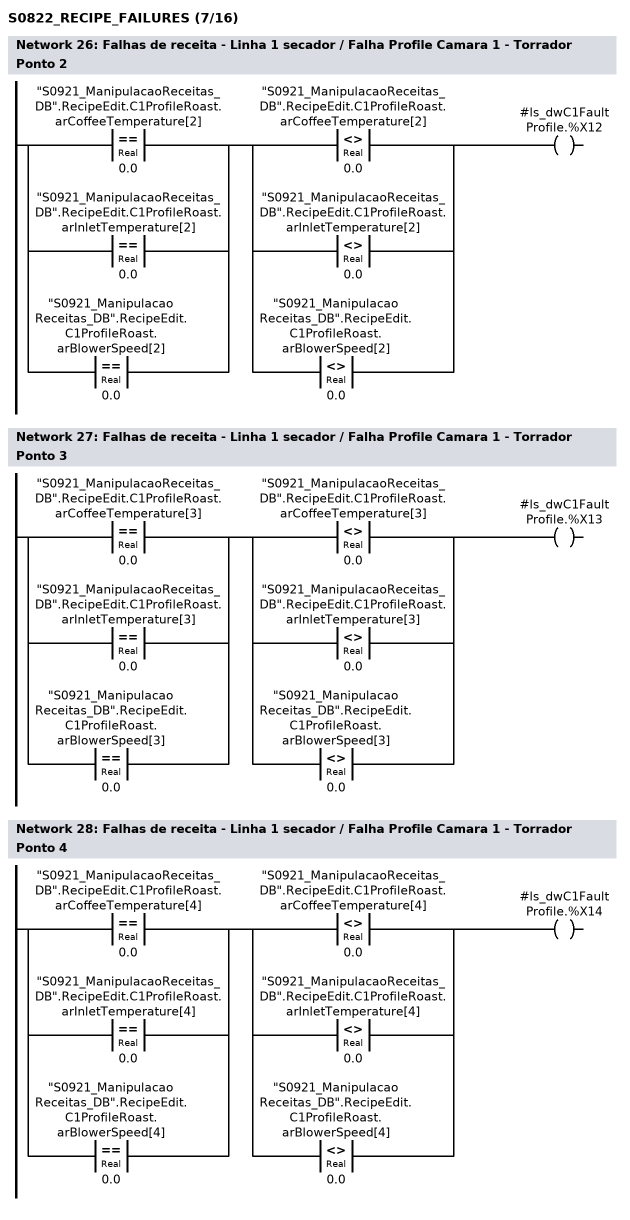
   RUNG wire#powerrail
      { S7_Templates := "SrcType := Real" } EQ_Contact(in1 := "S0921_ManipulacaoReceitas_DB".RecipeEdit.C1ProfileRoast.arCoffeeTemperature[2], in2 := 0.0)
      wire#w1
      { S7_Templates := "SrcType := Real" } NE_Contact(in1 := "S0921_ManipulacaoReceitas_DB".RecipeEdit.C1ProfileRoast.arCoffeeTemperature[2], in2 := 0.0)
      wire#w2
      Coil( #ls_dwC1FaultProfile.%X12 )
   END_RUNG
   RUNG wire#powerrail
      { S7_Templates := "SrcType := Real" } EQ_Contact(in1 := "S0921_ManipulacaoReceitas_DB".RecipeEdit.C1ProfileRoast.arInletTemperature[2], in2 := 0.0)
   END_RUNG wire#w1
   RUNG wire#powerrail
      { S7_Templates := "SrcType := Real" } EQ_Contact(in1 := "S0921_ManipulacaoReceitas_DB".RecipeEdit.C1ProfileRoast.arBlowerSpeed[2], in2 := 0.0)
   END_RUNG wire#w1
   RUNG wire#w1
      { S7_Templates := "SrcType := Real" } NE_Contact(in1 := "S0921_ManipulacaoReceitas_DB".RecipeEdit.C1ProfileRoast.arInletTemperature[2], in2 := 0.0)
   END_RUNG wire#w2
   RUNG wire#w1
      { S7_Templates := "SrcType := Real" } NE_Contact(in1 := "S0921_ManipulacaoReceitas_DB".RecipeEdit.C1ProfileRoast.arBlowerSpeed[2], in2 := 0.0)
   END_RUNG wire#w2
   // the same network as SCL:
   #ls_dwC1FaultProfile.%X12 := (("S0921_ManipulacaoReceitas_DB".RecipeEdit.C1ProfileRoast.arCoffeeTemperature[2] = 0.0) OR ("S0921_ManipulacaoReceitas_DB".RecipeEdit.C1ProfileRoast.arInletTemperature[2] = 0.0) OR ("S0921_ManipulacaoReceitas_DB".RecipeEdit.C1ProfileRoast.arBlowerSpeed[2] = 0.0)) AND (("S0921_ManipulacaoReceitas_DB".RecipeEdit.C1ProfileRoast.arCoffeeTemperature[2] <> 0.0) OR ("S0921_ManipulacaoReceitas_DB".RecipeEdit.C1ProfileRoast.arInletTemperature[2] <> 0.0) OR ("S0921_ManipulacaoReceitas_DB".RecipeEdit.C1ProfileRoast.arBlowerSpeed[2] <> 0.0));
END_REGION

REGION Network 27: Falhas de receita - Linha 1 secador / Falha Profile Camara 1 - Torrador Ponto 3
   RUNG wire#powerrail
      { S7_Templates := "SrcType := Real" } EQ_Contact(in1 := "S0921_ManipulacaoReceitas_DB".RecipeEdit.C1ProfileRoast.arCoffeeTemperature[3], in2 := 0.0)
      wire#w1
      { S7_Templates := "SrcType := Real" } NE_Contact(in1 := "S0921_ManipulacaoReceitas_DB".RecipeEdit.C1ProfileRoast.arCoffeeTemperature[3], in2 := 0.0)
      wire#w2
      Coil( #ls_dwC1FaultProfile.%X13 )
   END_RUNG
   RUNG wire#powerrail
      { S7_Templates := "SrcType := Real" } EQ_Contact(in1 := "S0921_ManipulacaoReceitas_DB".RecipeEdit.C1ProfileRoast.arInletTemperature[3], in2 := 0.0)
   END_RUNG wire#w1
   RUNG wire#powerrail
      { S7_Templates := "SrcType := Real" } EQ_Contact(in1 := "S0921_ManipulacaoReceitas_DB".RecipeEdit.C1ProfileRoast.arBlowerSpeed[3], in2 := 0.0)
   END_RUNG wire#w1
   RUNG wire#w1
      { S7_Templates := "SrcType := Real" } NE_Contact(in1 := "S0921_ManipulacaoReceitas_DB".RecipeEdit.C1ProfileRoast.arInletTemperature[3], in2 := 0.0)
   END_RUNG wire#w2
   RUNG wire#w1
      { S7_Templates := "SrcType := Real" } NE_Contact(in1 := "S0921_ManipulacaoReceitas_DB".RecipeEdit.C1ProfileRoast.arBlowerSpeed[3], in2 := 0.0)
   END_RUNG wire#w2
   // the same network as SCL:
   #ls_dwC1FaultProfile.%X13 := (("S0921_ManipulacaoReceitas_DB".RecipeEdit.C1ProfileRoast.arCoffeeTemperature[3] = 0.0) OR ("S0921_ManipulacaoReceitas_DB".RecipeEdit.C1ProfileRoast.arInletTemperature[3] = 0.0) OR ("S0921_ManipulacaoReceitas_DB".RecipeEdit.C1ProfileRoast.arBlowerSpeed[3] = 0.0)) AND (("S0921_ManipulacaoReceitas_DB".RecipeEdit.C1ProfileRoast.arCoffeeTemperature[3] <> 0.0) OR ("S0921_ManipulacaoReceitas_DB".RecipeEdit.C1ProfileRoast.arInletTemperature[3] <> 0.0) OR ("S0921_ManipulacaoReceitas_DB".RecipeEdit.C1ProfileRoast.arBlowerSpeed[3] <> 0.0));
END_REGION

REGION Network 28: Falhas de receita - Linha 1 secador / Falha Profile Camara 1 - Torrador Ponto 4
   RUNG wire#powerrail
      { S7_Templates := "SrcType := Real" } EQ_Contact(in1 := "S0921_ManipulacaoReceitas_DB".RecipeEdit.C1ProfileRoast.arCoffeeTemperature[4], in2 := 0.0)
      wire#w1
      { S7_Templates := "SrcType := Real" } NE_Contact(in1 := "S0921_ManipulacaoReceitas_DB".RecipeEdit.C1ProfileRoast.arCoffeeTemperature[4], in2 := 0.0)
      wire#w2
      Coil( #ls_dwC1FaultProfile.%X14 )
   END_RUNG
   RUNG wire#powerrail
      { S7_Templates := "SrcType := Real" } EQ_Contact(in1 := "S0921_ManipulacaoReceitas_DB".RecipeEdit.C1ProfileRoast.arInletTemperature[4], in2 := 0.0)
   END_RUNG wire#w1
   RUNG wire#powerrail
      { S7_Templates := "SrcType := Real" } EQ_Contact(in1 := "S0921_ManipulacaoReceitas_DB".RecipeEdit.C1ProfileRoast.arBlowerSpeed[4], in2 := 0.0)
   END_RUNG wire#w1
   RUNG wire#w1
      { S7_Templates := "SrcType := Real" } NE_Contact(in1 := "S0921_ManipulacaoReceitas_DB".RecipeEdit.C1ProfileRoast.arInletTemperature[4], in2 := 0.0)
   END_RUNG wire#w2
   RUNG wire#w1
      { S7_Templates := "SrcType := Real" } NE_Contact(in1 := "S0921_ManipulacaoReceitas_DB".RecipeEdit.C1ProfileRoast.arBlowerSpeed[4], in2 := 0.0)
   END_RUNG wire#w2
   // the same network as SCL:
   #ls_dwC1FaultProfile.%X14 := (("S0921_ManipulacaoReceitas_DB".RecipeEdit.C1ProfileRoast.arCoffeeTemperature[4] = 0.0) OR ("S0921_ManipulacaoReceitas_DB".RecipeEdit.C1ProfileRoast.arInletTemperature[4] = 0.0) OR ("S0921_ManipulacaoReceitas_DB".RecipeEdit.C1ProfileRoast.arBlowerSpeed[4] = 0.0)) AND (("S0921_ManipulacaoReceitas_DB".RecipeEdit.C1ProfileRoast.arCoffeeTemperature[4] <> 0.0) OR ("S0921_ManipulacaoReceitas_DB".RecipeEdit.C1ProfileRoast.arInletTemperature[4] <> 0.0) OR ("S0921_ManipulacaoReceitas_DB".RecipeEdit.C1ProfileRoast.arBlowerSpeed[4] <> 0.0));
END_REGION

REGION Network 29: Falhas de receita - Linha 1 secador / Falha Profile Camara 1 - Torrador Ponto 5
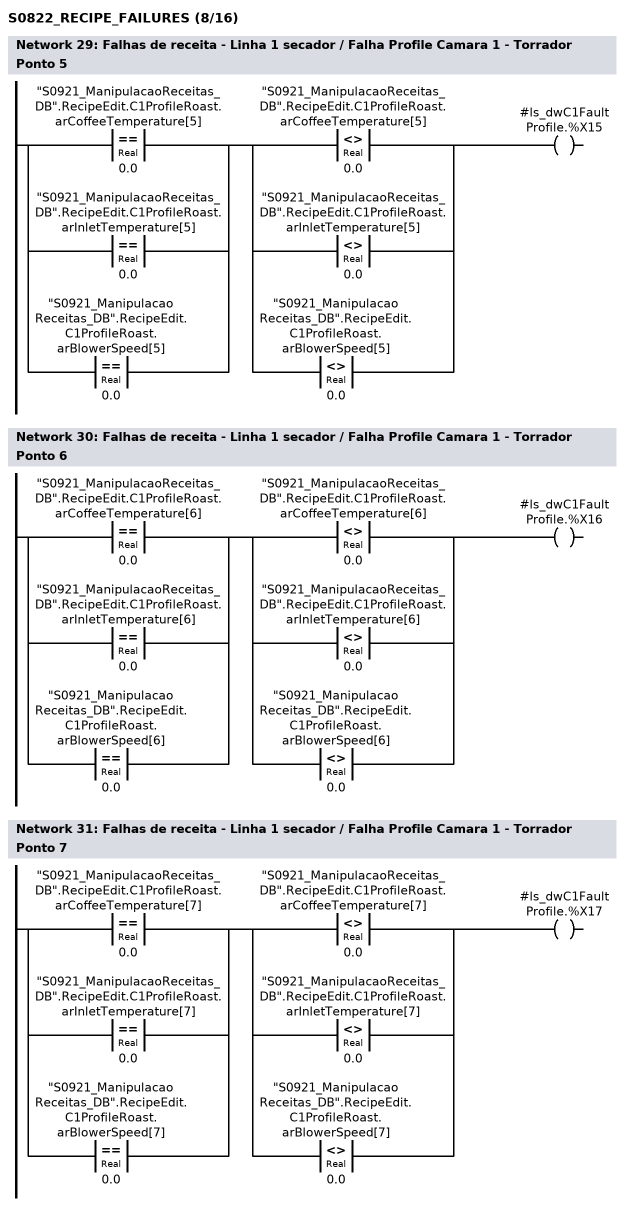
   RUNG wire#powerrail
      { S7_Templates := "SrcType := Real" } EQ_Contact(in1 := "S0921_ManipulacaoReceitas_DB".RecipeEdit.C1ProfileRoast.arCoffeeTemperature[5], in2 := 0.0)
      wire#w1
      { S7_Templates := "SrcType := Real" } NE_Contact(in1 := "S0921_ManipulacaoReceitas_DB".RecipeEdit.C1ProfileRoast.arCoffeeTemperature[5], in2 := 0.0)
      wire#w2
      Coil( #ls_dwC1FaultProfile.%X15 )
   END_RUNG
   RUNG wire#powerrail
      { S7_Templates := "SrcType := Real" } EQ_Contact(in1 := "S0921_ManipulacaoReceitas_DB".RecipeEdit.C1ProfileRoast.arInletTemperature[5], in2 := 0.0)
   END_RUNG wire#w1
   RUNG wire#powerrail
      { S7_Templates := "SrcType := Real" } EQ_Contact(in1 := "S0921_ManipulacaoReceitas_DB".RecipeEdit.C1ProfileRoast.arBlowerSpeed[5], in2 := 0.0)
   END_RUNG wire#w1
   RUNG wire#w1
      { S7_Templates := "SrcType := Real" } NE_Contact(in1 := "S0921_ManipulacaoReceitas_DB".RecipeEdit.C1ProfileRoast.arInletTemperature[5], in2 := 0.0)
   END_RUNG wire#w2
   RUNG wire#w1
      { S7_Templates := "SrcType := Real" } NE_Contact(in1 := "S0921_ManipulacaoReceitas_DB".RecipeEdit.C1ProfileRoast.arBlowerSpeed[5], in2 := 0.0)
   END_RUNG wire#w2
   // the same network as SCL:
   #ls_dwC1FaultProfile.%X15 := (("S0921_ManipulacaoReceitas_DB".RecipeEdit.C1ProfileRoast.arCoffeeTemperature[5] = 0.0) OR ("S0921_ManipulacaoReceitas_DB".RecipeEdit.C1ProfileRoast.arInletTemperature[5] = 0.0) OR ("S0921_ManipulacaoReceitas_DB".RecipeEdit.C1ProfileRoast.arBlowerSpeed[5] = 0.0)) AND (("S0921_ManipulacaoReceitas_DB".RecipeEdit.C1ProfileRoast.arCoffeeTemperature[5] <> 0.0) OR ("S0921_ManipulacaoReceitas_DB".RecipeEdit.C1ProfileRoast.arInletTemperature[5] <> 0.0) OR ("S0921_ManipulacaoReceitas_DB".RecipeEdit.C1ProfileRoast.arBlowerSpeed[5] <> 0.0));
END_REGION

REGION Network 30: Falhas de receita - Linha 1 secador / Falha Profile Camara 1 - Torrador Ponto 6
   RUNG wire#powerrail
      { S7_Templates := "SrcType := Real" } EQ_Contact(in1 := "S0921_ManipulacaoReceitas_DB".RecipeEdit.C1ProfileRoast.arCoffeeTemperature[6], in2 := 0.0)
      wire#w1
      { S7_Templates := "SrcType := Real" } NE_Contact(in1 := "S0921_ManipulacaoReceitas_DB".RecipeEdit.C1ProfileRoast.arCoffeeTemperature[6], in2 := 0.0)
      wire#w2
      Coil( #ls_dwC1FaultProfile.%X16 )
   END_RUNG
   RUNG wire#powerrail
      { S7_Templates := "SrcType := Real" } EQ_Contact(in1 := "S0921_ManipulacaoReceitas_DB".RecipeEdit.C1ProfileRoast.arInletTemperature[6], in2 := 0.0)
   END_RUNG wire#w1
   RUNG wire#powerrail
      { S7_Templates := "SrcType := Real" } EQ_Contact(in1 := "S0921_ManipulacaoReceitas_DB".RecipeEdit.C1ProfileRoast.arBlowerSpeed[6], in2 := 0.0)
   END_RUNG wire#w1
   RUNG wire#w1
      { S7_Templates := "SrcType := Real" } NE_Contact(in1 := "S0921_ManipulacaoReceitas_DB".RecipeEdit.C1ProfileRoast.arInletTemperature[6], in2 := 0.0)
   END_RUNG wire#w2
   RUNG wire#w1
      { S7_Templates := "SrcType := Real" } NE_Contact(in1 := "S0921_ManipulacaoReceitas_DB".RecipeEdit.C1ProfileRoast.arBlowerSpeed[6], in2 := 0.0)
   END_RUNG wire#w2
   // the same network as SCL:
   #ls_dwC1FaultProfile.%X16 := (("S0921_ManipulacaoReceitas_DB".RecipeEdit.C1ProfileRoast.arCoffeeTemperature[6] = 0.0) OR ("S0921_ManipulacaoReceitas_DB".RecipeEdit.C1ProfileRoast.arInletTemperature[6] = 0.0) OR ("S0921_ManipulacaoReceitas_DB".RecipeEdit.C1ProfileRoast.arBlowerSpeed[6] = 0.0)) AND (("S0921_ManipulacaoReceitas_DB".RecipeEdit.C1ProfileRoast.arCoffeeTemperature[6] <> 0.0) OR ("S0921_ManipulacaoReceitas_DB".RecipeEdit.C1ProfileRoast.arInletTemperature[6] <> 0.0) OR ("S0921_ManipulacaoReceitas_DB".RecipeEdit.C1ProfileRoast.arBlowerSpeed[6] <> 0.0));
END_REGION

REGION Network 31: Falhas de receita - Linha 1 secador / Falha Profile Camara 1 - Torrador Ponto 7
   RUNG wire#powerrail
      { S7_Templates := "SrcType := Real" } EQ_Contact(in1 := "S0921_ManipulacaoReceitas_DB".RecipeEdit.C1ProfileRoast.arCoffeeTemperature[7], in2 := 0.0)
      wire#w1
      { S7_Templates := "SrcType := Real" } NE_Contact(in1 := "S0921_ManipulacaoReceitas_DB".RecipeEdit.C1ProfileRoast.arCoffeeTemperature[7], in2 := 0.0)
      wire#w2
      Coil( #ls_dwC1FaultProfile.%X17 )
   END_RUNG
   RUNG wire#powerrail
      { S7_Templates := "SrcType := Real" } EQ_Contact(in1 := "S0921_ManipulacaoReceitas_DB".RecipeEdit.C1ProfileRoast.arInletTemperature[7], in2 := 0.0)
   END_RUNG wire#w1
   RUNG wire#powerrail
      { S7_Templates := "SrcType := Real" } EQ_Contact(in1 := "S0921_ManipulacaoReceitas_DB".RecipeEdit.C1ProfileRoast.arBlowerSpeed[7], in2 := 0.0)
   END_RUNG wire#w1
   RUNG wire#w1
      { S7_Templates := "SrcType := Real" } NE_Contact(in1 := "S0921_ManipulacaoReceitas_DB".RecipeEdit.C1ProfileRoast.arInletTemperature[7], in2 := 0.0)
   END_RUNG wire#w2
   RUNG wire#w1
      { S7_Templates := "SrcType := Real" } NE_Contact(in1 := "S0921_ManipulacaoReceitas_DB".RecipeEdit.C1ProfileRoast.arBlowerSpeed[7], in2 := 0.0)
   END_RUNG wire#w2
   // the same network as SCL:
   #ls_dwC1FaultProfile.%X17 := (("S0921_ManipulacaoReceitas_DB".RecipeEdit.C1ProfileRoast.arCoffeeTemperature[7] = 0.0) OR ("S0921_ManipulacaoReceitas_DB".RecipeEdit.C1ProfileRoast.arInletTemperature[7] = 0.0) OR ("S0921_ManipulacaoReceitas_DB".RecipeEdit.C1ProfileRoast.arBlowerSpeed[7] = 0.0)) AND (("S0921_ManipulacaoReceitas_DB".RecipeEdit.C1ProfileRoast.arCoffeeTemperature[7] <> 0.0) OR ("S0921_ManipulacaoReceitas_DB".RecipeEdit.C1ProfileRoast.arInletTemperature[7] <> 0.0) OR ("S0921_ManipulacaoReceitas_DB".RecipeEdit.C1ProfileRoast.arBlowerSpeed[7] <> 0.0));
END_REGION

REGION Network 32: Falhas de receita - Linha 1 secador / Falha Profile Camara 1 - Torrador Ponto 8
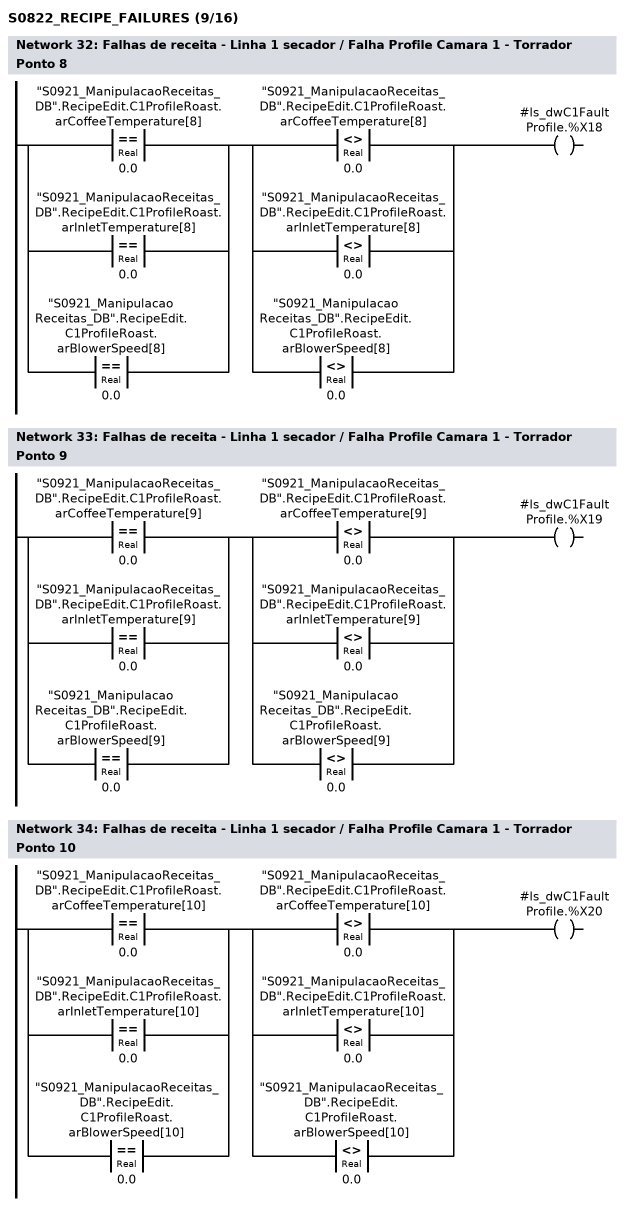
   RUNG wire#powerrail
      { S7_Templates := "SrcType := Real" } EQ_Contact(in1 := "S0921_ManipulacaoReceitas_DB".RecipeEdit.C1ProfileRoast.arCoffeeTemperature[8], in2 := 0.0)
      wire#w1
      { S7_Templates := "SrcType := Real" } NE_Contact(in1 := "S0921_ManipulacaoReceitas_DB".RecipeEdit.C1ProfileRoast.arCoffeeTemperature[8], in2 := 0.0)
      wire#w2
      Coil( #ls_dwC1FaultProfile.%X18 )
   END_RUNG
   RUNG wire#powerrail
      { S7_Templates := "SrcType := Real" } EQ_Contact(in1 := "S0921_ManipulacaoReceitas_DB".RecipeEdit.C1ProfileRoast.arInletTemperature[8], in2 := 0.0)
   END_RUNG wire#w1
   RUNG wire#powerrail
      { S7_Templates := "SrcType := Real" } EQ_Contact(in1 := "S0921_ManipulacaoReceitas_DB".RecipeEdit.C1ProfileRoast.arBlowerSpeed[8], in2 := 0.0)
   END_RUNG wire#w1
   RUNG wire#w1
      { S7_Templates := "SrcType := Real" } NE_Contact(in1 := "S0921_ManipulacaoReceitas_DB".RecipeEdit.C1ProfileRoast.arInletTemperature[8], in2 := 0.0)
   END_RUNG wire#w2
   RUNG wire#w1
      { S7_Templates := "SrcType := Real" } NE_Contact(in1 := "S0921_ManipulacaoReceitas_DB".RecipeEdit.C1ProfileRoast.arBlowerSpeed[8], in2 := 0.0)
   END_RUNG wire#w2
   // the same network as SCL:
   #ls_dwC1FaultProfile.%X18 := (("S0921_ManipulacaoReceitas_DB".RecipeEdit.C1ProfileRoast.arCoffeeTemperature[8] = 0.0) OR ("S0921_ManipulacaoReceitas_DB".RecipeEdit.C1ProfileRoast.arInletTemperature[8] = 0.0) OR ("S0921_ManipulacaoReceitas_DB".RecipeEdit.C1ProfileRoast.arBlowerSpeed[8] = 0.0)) AND (("S0921_ManipulacaoReceitas_DB".RecipeEdit.C1ProfileRoast.arCoffeeTemperature[8] <> 0.0) OR ("S0921_ManipulacaoReceitas_DB".RecipeEdit.C1ProfileRoast.arInletTemperature[8] <> 0.0) OR ("S0921_ManipulacaoReceitas_DB".RecipeEdit.C1ProfileRoast.arBlowerSpeed[8] <> 0.0));
END_REGION

REGION Network 33: Falhas de receita - Linha 1 secador / Falha Profile Camara 1 - Torrador Ponto 9
   RUNG wire#powerrail
      { S7_Templates := "SrcType := Real" } EQ_Contact(in1 := "S0921_ManipulacaoReceitas_DB".RecipeEdit.C1ProfileRoast.arCoffeeTemperature[9], in2 := 0.0)
      wire#w1
      { S7_Templates := "SrcType := Real" } NE_Contact(in1 := "S0921_ManipulacaoReceitas_DB".RecipeEdit.C1ProfileRoast.arCoffeeTemperature[9], in2 := 0.0)
      wire#w2
      Coil( #ls_dwC1FaultProfile.%X19 )
   END_RUNG
   RUNG wire#powerrail
      { S7_Templates := "SrcType := Real" } EQ_Contact(in1 := "S0921_ManipulacaoReceitas_DB".RecipeEdit.C1ProfileRoast.arInletTemperature[9], in2 := 0.0)
   END_RUNG wire#w1
   RUNG wire#powerrail
      { S7_Templates := "SrcType := Real" } EQ_Contact(in1 := "S0921_ManipulacaoReceitas_DB".RecipeEdit.C1ProfileRoast.arBlowerSpeed[9], in2 := 0.0)
   END_RUNG wire#w1
   RUNG wire#w1
      { S7_Templates := "SrcType := Real" } NE_Contact(in1 := "S0921_ManipulacaoReceitas_DB".RecipeEdit.C1ProfileRoast.arInletTemperature[9], in2 := 0.0)
   END_RUNG wire#w2
   RUNG wire#w1
      { S7_Templates := "SrcType := Real" } NE_Contact(in1 := "S0921_ManipulacaoReceitas_DB".RecipeEdit.C1ProfileRoast.arBlowerSpeed[9], in2 := 0.0)
   END_RUNG wire#w2
   // the same network as SCL:
   #ls_dwC1FaultProfile.%X19 := (("S0921_ManipulacaoReceitas_DB".RecipeEdit.C1ProfileRoast.arCoffeeTemperature[9] = 0.0) OR ("S0921_ManipulacaoReceitas_DB".RecipeEdit.C1ProfileRoast.arInletTemperature[9] = 0.0) OR ("S0921_ManipulacaoReceitas_DB".RecipeEdit.C1ProfileRoast.arBlowerSpeed[9] = 0.0)) AND (("S0921_ManipulacaoReceitas_DB".RecipeEdit.C1ProfileRoast.arCoffeeTemperature[9] <> 0.0) OR ("S0921_ManipulacaoReceitas_DB".RecipeEdit.C1ProfileRoast.arInletTemperature[9] <> 0.0) OR ("S0921_ManipulacaoReceitas_DB".RecipeEdit.C1ProfileRoast.arBlowerSpeed[9] <> 0.0));
END_REGION

REGION Network 34: Falhas de receita - Linha 1 secador / Falha Profile Camara 1 - Torrador Ponto 10
   RUNG wire#powerrail
      { S7_Templates := "SrcType := Real" } EQ_Contact(in1 := "S0921_ManipulacaoReceitas_DB".RecipeEdit.C1ProfileRoast.arCoffeeTemperature[10], in2 := 0.0)
      wire#w1
      { S7_Templates := "SrcType := Real" } NE_Contact(in1 := "S0921_ManipulacaoReceitas_DB".RecipeEdit.C1ProfileRoast.arCoffeeTemperature[10], in2 := 0.0)
      wire#w2
      Coil( #ls_dwC1FaultProfile.%X20 )
   END_RUNG
   RUNG wire#powerrail
      { S7_Templates := "SrcType := Real" } EQ_Contact(in1 := "S0921_ManipulacaoReceitas_DB".RecipeEdit.C1ProfileRoast.arInletTemperature[10], in2 := 0.0)
   END_RUNG wire#w1
   RUNG wire#powerrail
      { S7_Templates := "SrcType := Real" } EQ_Contact(in1 := "S0921_ManipulacaoReceitas_DB".RecipeEdit.C1ProfileRoast.arBlowerSpeed[10], in2 := 0.0)
   END_RUNG wire#w1
   RUNG wire#w1
      { S7_Templates := "SrcType := Real" } NE_Contact(in1 := "S0921_ManipulacaoReceitas_DB".RecipeEdit.C1ProfileRoast.arInletTemperature[10], in2 := 0.0)
   END_RUNG wire#w2
   RUNG wire#w1
      { S7_Templates := "SrcType := Real" } NE_Contact(in1 := "S0921_ManipulacaoReceitas_DB".RecipeEdit.C1ProfileRoast.arBlowerSpeed[10], in2 := 0.0)
   END_RUNG wire#w2
   // the same network as SCL:
   #ls_dwC1FaultProfile.%X20 := (("S0921_ManipulacaoReceitas_DB".RecipeEdit.C1ProfileRoast.arCoffeeTemperature[10] = 0.0) OR ("S0921_ManipulacaoReceitas_DB".RecipeEdit.C1ProfileRoast.arInletTemperature[10] = 0.0) OR ("S0921_ManipulacaoReceitas_DB".RecipeEdit.C1ProfileRoast.arBlowerSpeed[10] = 0.0)) AND (("S0921_ManipulacaoReceitas_DB".RecipeEdit.C1ProfileRoast.arCoffeeTemperature[10] <> 0.0) OR ("S0921_ManipulacaoReceitas_DB".RecipeEdit.C1ProfileRoast.arInletTemperature[10] <> 0.0) OR ("S0921_ManipulacaoReceitas_DB".RecipeEdit.C1ProfileRoast.arBlowerSpeed[10] <> 0.0));
END_REGION

REGION Network 35: Falhas de receita - Linha 1 secador / Falha Profile Camara 2 - Secador Ponto 1
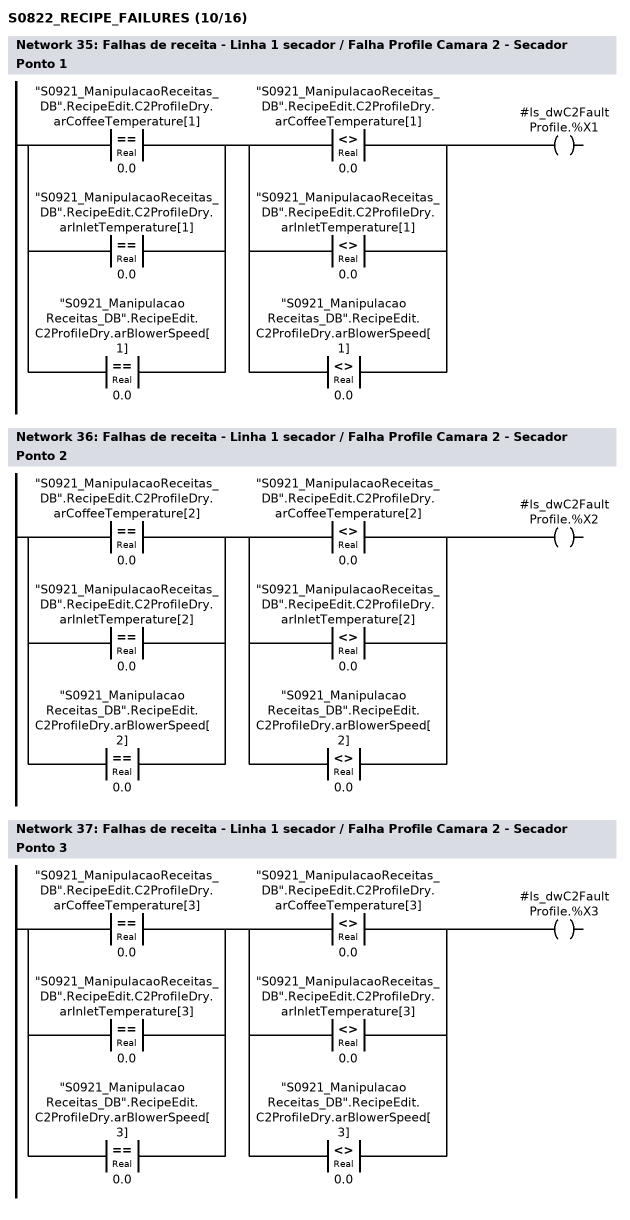
   RUNG wire#powerrail
      { S7_Templates := "SrcType := Real" } EQ_Contact(in1 := "S0921_ManipulacaoReceitas_DB".RecipeEdit.C2ProfileDry.arCoffeeTemperature[1], in2 := 0.0)
      wire#w1
      { S7_Templates := "SrcType := Real" } NE_Contact(in1 := "S0921_ManipulacaoReceitas_DB".RecipeEdit.C2ProfileDry.arCoffeeTemperature[1], in2 := 0.0)
      wire#w2
      Coil( #ls_dwC2FaultProfile.%X1 )
   END_RUNG
   RUNG wire#powerrail
      { S7_Templates := "SrcType := Real" } EQ_Contact(in1 := "S0921_ManipulacaoReceitas_DB".RecipeEdit.C2ProfileDry.arInletTemperature[1], in2 := 0.0)
   END_RUNG wire#w1
   RUNG wire#powerrail
      { S7_Templates := "SrcType := Real" } EQ_Contact(in1 := "S0921_ManipulacaoReceitas_DB".RecipeEdit.C2ProfileDry.arBlowerSpeed[1], in2 := 0.0)
   END_RUNG wire#w1
   RUNG wire#w1
      { S7_Templates := "SrcType := Real" } NE_Contact(in1 := "S0921_ManipulacaoReceitas_DB".RecipeEdit.C2ProfileDry.arInletTemperature[1], in2 := 0.0)
   END_RUNG wire#w2
   RUNG wire#w1
      { S7_Templates := "SrcType := Real" } NE_Contact(in1 := "S0921_ManipulacaoReceitas_DB".RecipeEdit.C2ProfileDry.arBlowerSpeed[1], in2 := 0.0)
   END_RUNG wire#w2
   // the same network as SCL:
   #ls_dwC2FaultProfile.%X1 := (("S0921_ManipulacaoReceitas_DB".RecipeEdit.C2ProfileDry.arCoffeeTemperature[1] = 0.0) OR ("S0921_ManipulacaoReceitas_DB".RecipeEdit.C2ProfileDry.arInletTemperature[1] = 0.0) OR ("S0921_ManipulacaoReceitas_DB".RecipeEdit.C2ProfileDry.arBlowerSpeed[1] = 0.0)) AND (("S0921_ManipulacaoReceitas_DB".RecipeEdit.C2ProfileDry.arCoffeeTemperature[1] <> 0.0) OR ("S0921_ManipulacaoReceitas_DB".RecipeEdit.C2ProfileDry.arInletTemperature[1] <> 0.0) OR ("S0921_ManipulacaoReceitas_DB".RecipeEdit.C2ProfileDry.arBlowerSpeed[1] <> 0.0));
END_REGION

REGION Network 36: Falhas de receita - Linha 1 secador / Falha Profile Camara 2 - Secador Ponto 2
   RUNG wire#powerrail
      { S7_Templates := "SrcType := Real" } EQ_Contact(in1 := "S0921_ManipulacaoReceitas_DB".RecipeEdit.C2ProfileDry.arCoffeeTemperature[2], in2 := 0.0)
      wire#w1
      { S7_Templates := "SrcType := Real" } NE_Contact(in1 := "S0921_ManipulacaoReceitas_DB".RecipeEdit.C2ProfileDry.arCoffeeTemperature[2], in2 := 0.0)
      wire#w2
      Coil( #ls_dwC2FaultProfile.%X2 )
   END_RUNG
   RUNG wire#powerrail
      { S7_Templates := "SrcType := Real" } EQ_Contact(in1 := "S0921_ManipulacaoReceitas_DB".RecipeEdit.C2ProfileDry.arInletTemperature[2], in2 := 0.0)
   END_RUNG wire#w1
   RUNG wire#powerrail
      { S7_Templates := "SrcType := Real" } EQ_Contact(in1 := "S0921_ManipulacaoReceitas_DB".RecipeEdit.C2ProfileDry.arBlowerSpeed[2], in2 := 0.0)
   END_RUNG wire#w1
   RUNG wire#w1
      { S7_Templates := "SrcType := Real" } NE_Contact(in1 := "S0921_ManipulacaoReceitas_DB".RecipeEdit.C2ProfileDry.arInletTemperature[2], in2 := 0.0)
   END_RUNG wire#w2
   RUNG wire#w1
      { S7_Templates := "SrcType := Real" } NE_Contact(in1 := "S0921_ManipulacaoReceitas_DB".RecipeEdit.C2ProfileDry.arBlowerSpeed[2], in2 := 0.0)
   END_RUNG wire#w2
   // the same network as SCL:
   #ls_dwC2FaultProfile.%X2 := (("S0921_ManipulacaoReceitas_DB".RecipeEdit.C2ProfileDry.arCoffeeTemperature[2] = 0.0) OR ("S0921_ManipulacaoReceitas_DB".RecipeEdit.C2ProfileDry.arInletTemperature[2] = 0.0) OR ("S0921_ManipulacaoReceitas_DB".RecipeEdit.C2ProfileDry.arBlowerSpeed[2] = 0.0)) AND (("S0921_ManipulacaoReceitas_DB".RecipeEdit.C2ProfileDry.arCoffeeTemperature[2] <> 0.0) OR ("S0921_ManipulacaoReceitas_DB".RecipeEdit.C2ProfileDry.arInletTemperature[2] <> 0.0) OR ("S0921_ManipulacaoReceitas_DB".RecipeEdit.C2ProfileDry.arBlowerSpeed[2] <> 0.0));
END_REGION

REGION Network 37: Falhas de receita - Linha 1 secador / Falha Profile Camara 2 - Secador Ponto 3
   RUNG wire#powerrail
      { S7_Templates := "SrcType := Real" } EQ_Contact(in1 := "S0921_ManipulacaoReceitas_DB".RecipeEdit.C2ProfileDry.arCoffeeTemperature[3], in2 := 0.0)
      wire#w1
      { S7_Templates := "SrcType := Real" } NE_Contact(in1 := "S0921_ManipulacaoReceitas_DB".RecipeEdit.C2ProfileDry.arCoffeeTemperature[3], in2 := 0.0)
      wire#w2
      Coil( #ls_dwC2FaultProfile.%X3 )
   END_RUNG
   RUNG wire#powerrail
      { S7_Templates := "SrcType := Real" } EQ_Contact(in1 := "S0921_ManipulacaoReceitas_DB".RecipeEdit.C2ProfileDry.arInletTemperature[3], in2 := 0.0)
   END_RUNG wire#w1
   RUNG wire#powerrail
      { S7_Templates := "SrcType := Real" } EQ_Contact(in1 := "S0921_ManipulacaoReceitas_DB".RecipeEdit.C2ProfileDry.arBlowerSpeed[3], in2 := 0.0)
   END_RUNG wire#w1
   RUNG wire#w1
      { S7_Templates := "SrcType := Real" } NE_Contact(in1 := "S0921_ManipulacaoReceitas_DB".RecipeEdit.C2ProfileDry.arInletTemperature[3], in2 := 0.0)
   END_RUNG wire#w2
   RUNG wire#w1
      { S7_Templates := "SrcType := Real" } NE_Contact(in1 := "S0921_ManipulacaoReceitas_DB".RecipeEdit.C2ProfileDry.arBlowerSpeed[3], in2 := 0.0)
   END_RUNG wire#w2
   // the same network as SCL:
   #ls_dwC2FaultProfile.%X3 := (("S0921_ManipulacaoReceitas_DB".RecipeEdit.C2ProfileDry.arCoffeeTemperature[3] = 0.0) OR ("S0921_ManipulacaoReceitas_DB".RecipeEdit.C2ProfileDry.arInletTemperature[3] = 0.0) OR ("S0921_ManipulacaoReceitas_DB".RecipeEdit.C2ProfileDry.arBlowerSpeed[3] = 0.0)) AND (("S0921_ManipulacaoReceitas_DB".RecipeEdit.C2ProfileDry.arCoffeeTemperature[3] <> 0.0) OR ("S0921_ManipulacaoReceitas_DB".RecipeEdit.C2ProfileDry.arInletTemperature[3] <> 0.0) OR ("S0921_ManipulacaoReceitas_DB".RecipeEdit.C2ProfileDry.arBlowerSpeed[3] <> 0.0));
END_REGION

REGION Network 38: Falhas de receita - Linha 1 secador / Falha Profile Camara 2 - Secador Ponto 4
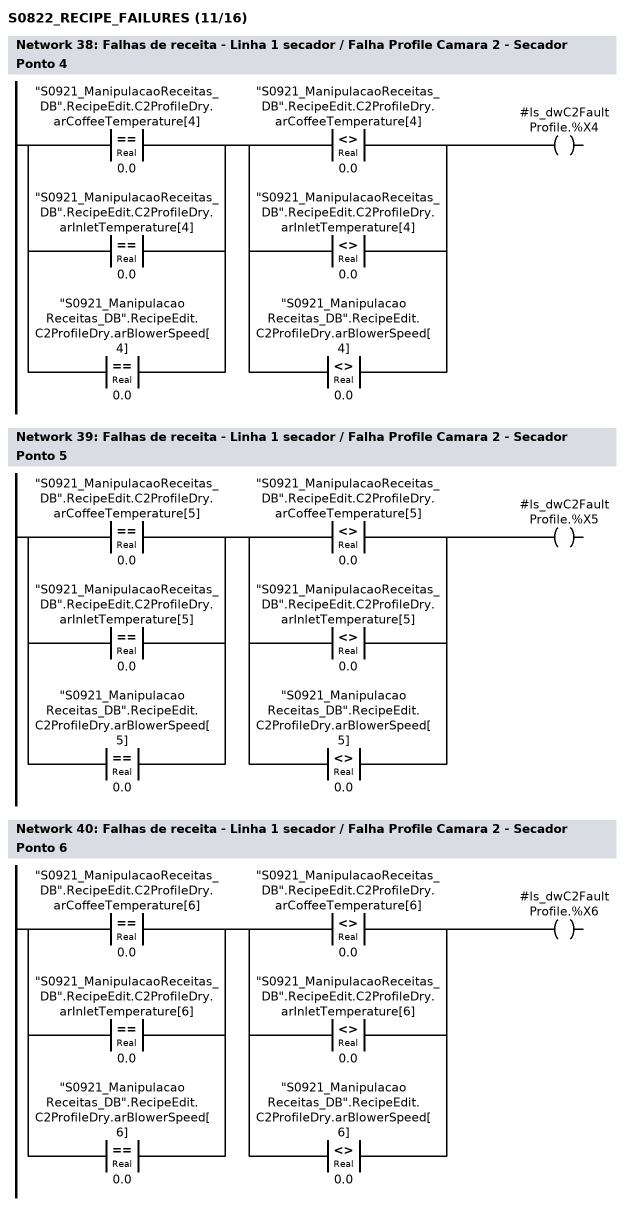
   RUNG wire#powerrail
      { S7_Templates := "SrcType := Real" } EQ_Contact(in1 := "S0921_ManipulacaoReceitas_DB".RecipeEdit.C2ProfileDry.arCoffeeTemperature[4], in2 := 0.0)
      wire#w1
      { S7_Templates := "SrcType := Real" } NE_Contact(in1 := "S0921_ManipulacaoReceitas_DB".RecipeEdit.C2ProfileDry.arCoffeeTemperature[4], in2 := 0.0)
      wire#w2
      Coil( #ls_dwC2FaultProfile.%X4 )
   END_RUNG
   RUNG wire#powerrail
      { S7_Templates := "SrcType := Real" } EQ_Contact(in1 := "S0921_ManipulacaoReceitas_DB".RecipeEdit.C2ProfileDry.arInletTemperature[4], in2 := 0.0)
   END_RUNG wire#w1
   RUNG wire#powerrail
      { S7_Templates := "SrcType := Real" } EQ_Contact(in1 := "S0921_ManipulacaoReceitas_DB".RecipeEdit.C2ProfileDry.arBlowerSpeed[4], in2 := 0.0)
   END_RUNG wire#w1
   RUNG wire#w1
      { S7_Templates := "SrcType := Real" } NE_Contact(in1 := "S0921_ManipulacaoReceitas_DB".RecipeEdit.C2ProfileDry.arInletTemperature[4], in2 := 0.0)
   END_RUNG wire#w2
   RUNG wire#w1
      { S7_Templates := "SrcType := Real" } NE_Contact(in1 := "S0921_ManipulacaoReceitas_DB".RecipeEdit.C2ProfileDry.arBlowerSpeed[4], in2 := 0.0)
   END_RUNG wire#w2
   // the same network as SCL:
   #ls_dwC2FaultProfile.%X4 := (("S0921_ManipulacaoReceitas_DB".RecipeEdit.C2ProfileDry.arCoffeeTemperature[4] = 0.0) OR ("S0921_ManipulacaoReceitas_DB".RecipeEdit.C2ProfileDry.arInletTemperature[4] = 0.0) OR ("S0921_ManipulacaoReceitas_DB".RecipeEdit.C2ProfileDry.arBlowerSpeed[4] = 0.0)) AND (("S0921_ManipulacaoReceitas_DB".RecipeEdit.C2ProfileDry.arCoffeeTemperature[4] <> 0.0) OR ("S0921_ManipulacaoReceitas_DB".RecipeEdit.C2ProfileDry.arInletTemperature[4] <> 0.0) OR ("S0921_ManipulacaoReceitas_DB".RecipeEdit.C2ProfileDry.arBlowerSpeed[4] <> 0.0));
END_REGION

REGION Network 39: Falhas de receita - Linha 1 secador / Falha Profile Camara 2 - Secador Ponto 5
   RUNG wire#powerrail
      { S7_Templates := "SrcType := Real" } EQ_Contact(in1 := "S0921_ManipulacaoReceitas_DB".RecipeEdit.C2ProfileDry.arCoffeeTemperature[5], in2 := 0.0)
      wire#w1
      { S7_Templates := "SrcType := Real" } NE_Contact(in1 := "S0921_ManipulacaoReceitas_DB".RecipeEdit.C2ProfileDry.arCoffeeTemperature[5], in2 := 0.0)
      wire#w2
      Coil( #ls_dwC2FaultProfile.%X5 )
   END_RUNG
   RUNG wire#powerrail
      { S7_Templates := "SrcType := Real" } EQ_Contact(in1 := "S0921_ManipulacaoReceitas_DB".RecipeEdit.C2ProfileDry.arInletTemperature[5], in2 := 0.0)
   END_RUNG wire#w1
   RUNG wire#powerrail
      { S7_Templates := "SrcType := Real" } EQ_Contact(in1 := "S0921_ManipulacaoReceitas_DB".RecipeEdit.C2ProfileDry.arBlowerSpeed[5], in2 := 0.0)
   END_RUNG wire#w1
   RUNG wire#w1
      { S7_Templates := "SrcType := Real" } NE_Contact(in1 := "S0921_ManipulacaoReceitas_DB".RecipeEdit.C2ProfileDry.arInletTemperature[5], in2 := 0.0)
   END_RUNG wire#w2
   RUNG wire#w1
      { S7_Templates := "SrcType := Real" } NE_Contact(in1 := "S0921_ManipulacaoReceitas_DB".RecipeEdit.C2ProfileDry.arBlowerSpeed[5], in2 := 0.0)
   END_RUNG wire#w2
   // the same network as SCL:
   #ls_dwC2FaultProfile.%X5 := (("S0921_ManipulacaoReceitas_DB".RecipeEdit.C2ProfileDry.arCoffeeTemperature[5] = 0.0) OR ("S0921_ManipulacaoReceitas_DB".RecipeEdit.C2ProfileDry.arInletTemperature[5] = 0.0) OR ("S0921_ManipulacaoReceitas_DB".RecipeEdit.C2ProfileDry.arBlowerSpeed[5] = 0.0)) AND (("S0921_ManipulacaoReceitas_DB".RecipeEdit.C2ProfileDry.arCoffeeTemperature[5] <> 0.0) OR ("S0921_ManipulacaoReceitas_DB".RecipeEdit.C2ProfileDry.arInletTemperature[5] <> 0.0) OR ("S0921_ManipulacaoReceitas_DB".RecipeEdit.C2ProfileDry.arBlowerSpeed[5] <> 0.0));
END_REGION

REGION Network 40: Falhas de receita - Linha 1 secador / Falha Profile Camara 2 - Secador Ponto 6
   RUNG wire#powerrail
      { S7_Templates := "SrcType := Real" } EQ_Contact(in1 := "S0921_ManipulacaoReceitas_DB".RecipeEdit.C2ProfileDry.arCoffeeTemperature[6], in2 := 0.0)
      wire#w1
      { S7_Templates := "SrcType := Real" } NE_Contact(in1 := "S0921_ManipulacaoReceitas_DB".RecipeEdit.C2ProfileDry.arCoffeeTemperature[6], in2 := 0.0)
      wire#w2
      Coil( #ls_dwC2FaultProfile.%X6 )
   END_RUNG
   RUNG wire#powerrail
      { S7_Templates := "SrcType := Real" } EQ_Contact(in1 := "S0921_ManipulacaoReceitas_DB".RecipeEdit.C2ProfileDry.arInletTemperature[6], in2 := 0.0)
   END_RUNG wire#w1
   RUNG wire#powerrail
      { S7_Templates := "SrcType := Real" } EQ_Contact(in1 := "S0921_ManipulacaoReceitas_DB".RecipeEdit.C2ProfileDry.arBlowerSpeed[6], in2 := 0.0)
   END_RUNG wire#w1
   RUNG wire#w1
      { S7_Templates := "SrcType := Real" } NE_Contact(in1 := "S0921_ManipulacaoReceitas_DB".RecipeEdit.C2ProfileDry.arInletTemperature[6], in2 := 0.0)
   END_RUNG wire#w2
   RUNG wire#w1
      { S7_Templates := "SrcType := Real" } NE_Contact(in1 := "S0921_ManipulacaoReceitas_DB".RecipeEdit.C2ProfileDry.arBlowerSpeed[6], in2 := 0.0)
   END_RUNG wire#w2
   // the same network as SCL:
   #ls_dwC2FaultProfile.%X6 := (("S0921_ManipulacaoReceitas_DB".RecipeEdit.C2ProfileDry.arCoffeeTemperature[6] = 0.0) OR ("S0921_ManipulacaoReceitas_DB".RecipeEdit.C2ProfileDry.arInletTemperature[6] = 0.0) OR ("S0921_ManipulacaoReceitas_DB".RecipeEdit.C2ProfileDry.arBlowerSpeed[6] = 0.0)) AND (("S0921_ManipulacaoReceitas_DB".RecipeEdit.C2ProfileDry.arCoffeeTemperature[6] <> 0.0) OR ("S0921_ManipulacaoReceitas_DB".RecipeEdit.C2ProfileDry.arInletTemperature[6] <> 0.0) OR ("S0921_ManipulacaoReceitas_DB".RecipeEdit.C2ProfileDry.arBlowerSpeed[6] <> 0.0));
END_REGION

REGION Network 41: Falhas de receita - Linha 1 secador / Falha Profile Camara 2 - Secador Ponto 7
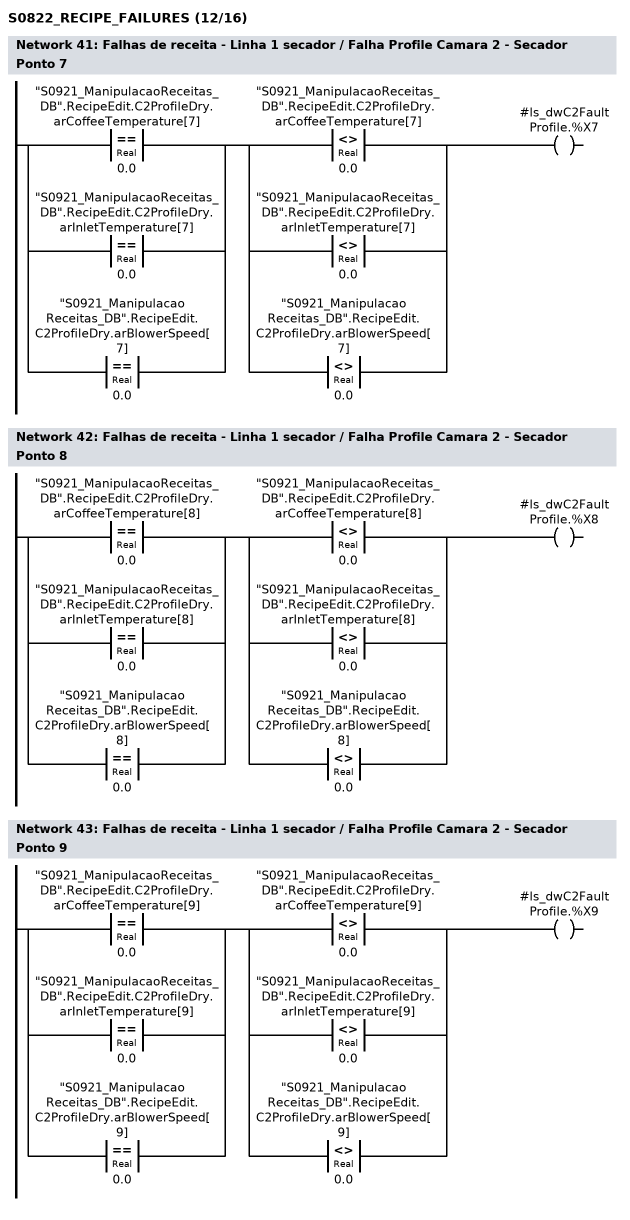
   RUNG wire#powerrail
      { S7_Templates := "SrcType := Real" } EQ_Contact(in1 := "S0921_ManipulacaoReceitas_DB".RecipeEdit.C2ProfileDry.arCoffeeTemperature[7], in2 := 0.0)
      wire#w1
      { S7_Templates := "SrcType := Real" } NE_Contact(in1 := "S0921_ManipulacaoReceitas_DB".RecipeEdit.C2ProfileDry.arCoffeeTemperature[7], in2 := 0.0)
      wire#w2
      Coil( #ls_dwC2FaultProfile.%X7 )
   END_RUNG
   RUNG wire#powerrail
      { S7_Templates := "SrcType := Real" } EQ_Contact(in1 := "S0921_ManipulacaoReceitas_DB".RecipeEdit.C2ProfileDry.arInletTemperature[7], in2 := 0.0)
   END_RUNG wire#w1
   RUNG wire#powerrail
      { S7_Templates := "SrcType := Real" } EQ_Contact(in1 := "S0921_ManipulacaoReceitas_DB".RecipeEdit.C2ProfileDry.arBlowerSpeed[7], in2 := 0.0)
   END_RUNG wire#w1
   RUNG wire#w1
      { S7_Templates := "SrcType := Real" } NE_Contact(in1 := "S0921_ManipulacaoReceitas_DB".RecipeEdit.C2ProfileDry.arInletTemperature[7], in2 := 0.0)
   END_RUNG wire#w2
   RUNG wire#w1
      { S7_Templates := "SrcType := Real" } NE_Contact(in1 := "S0921_ManipulacaoReceitas_DB".RecipeEdit.C2ProfileDry.arBlowerSpeed[7], in2 := 0.0)
   END_RUNG wire#w2
   // the same network as SCL:
   #ls_dwC2FaultProfile.%X7 := (("S0921_ManipulacaoReceitas_DB".RecipeEdit.C2ProfileDry.arCoffeeTemperature[7] = 0.0) OR ("S0921_ManipulacaoReceitas_DB".RecipeEdit.C2ProfileDry.arInletTemperature[7] = 0.0) OR ("S0921_ManipulacaoReceitas_DB".RecipeEdit.C2ProfileDry.arBlowerSpeed[7] = 0.0)) AND (("S0921_ManipulacaoReceitas_DB".RecipeEdit.C2ProfileDry.arCoffeeTemperature[7] <> 0.0) OR ("S0921_ManipulacaoReceitas_DB".RecipeEdit.C2ProfileDry.arInletTemperature[7] <> 0.0) OR ("S0921_ManipulacaoReceitas_DB".RecipeEdit.C2ProfileDry.arBlowerSpeed[7] <> 0.0));
END_REGION

REGION Network 42: Falhas de receita - Linha 1 secador / Falha Profile Camara 2 - Secador Ponto 8
   RUNG wire#powerrail
      { S7_Templates := "SrcType := Real" } EQ_Contact(in1 := "S0921_ManipulacaoReceitas_DB".RecipeEdit.C2ProfileDry.arCoffeeTemperature[8], in2 := 0.0)
      wire#w1
      { S7_Templates := "SrcType := Real" } NE_Contact(in1 := "S0921_ManipulacaoReceitas_DB".RecipeEdit.C2ProfileDry.arCoffeeTemperature[8], in2 := 0.0)
      wire#w2
      Coil( #ls_dwC2FaultProfile.%X8 )
   END_RUNG
   RUNG wire#powerrail
      { S7_Templates := "SrcType := Real" } EQ_Contact(in1 := "S0921_ManipulacaoReceitas_DB".RecipeEdit.C2ProfileDry.arInletTemperature[8], in2 := 0.0)
   END_RUNG wire#w1
   RUNG wire#powerrail
      { S7_Templates := "SrcType := Real" } EQ_Contact(in1 := "S0921_ManipulacaoReceitas_DB".RecipeEdit.C2ProfileDry.arBlowerSpeed[8], in2 := 0.0)
   END_RUNG wire#w1
   RUNG wire#w1
      { S7_Templates := "SrcType := Real" } NE_Contact(in1 := "S0921_ManipulacaoReceitas_DB".RecipeEdit.C2ProfileDry.arInletTemperature[8], in2 := 0.0)
   END_RUNG wire#w2
   RUNG wire#w1
      { S7_Templates := "SrcType := Real" } NE_Contact(in1 := "S0921_ManipulacaoReceitas_DB".RecipeEdit.C2ProfileDry.arBlowerSpeed[8], in2 := 0.0)
   END_RUNG wire#w2
   // the same network as SCL:
   #ls_dwC2FaultProfile.%X8 := (("S0921_ManipulacaoReceitas_DB".RecipeEdit.C2ProfileDry.arCoffeeTemperature[8] = 0.0) OR ("S0921_ManipulacaoReceitas_DB".RecipeEdit.C2ProfileDry.arInletTemperature[8] = 0.0) OR ("S0921_ManipulacaoReceitas_DB".RecipeEdit.C2ProfileDry.arBlowerSpeed[8] = 0.0)) AND (("S0921_ManipulacaoReceitas_DB".RecipeEdit.C2ProfileDry.arCoffeeTemperature[8] <> 0.0) OR ("S0921_ManipulacaoReceitas_DB".RecipeEdit.C2ProfileDry.arInletTemperature[8] <> 0.0) OR ("S0921_ManipulacaoReceitas_DB".RecipeEdit.C2ProfileDry.arBlowerSpeed[8] <> 0.0));
END_REGION

REGION Network 43: Falhas de receita - Linha 1 secador / Falha Profile Camara 2 - Secador Ponto 9
   RUNG wire#powerrail
      { S7_Templates := "SrcType := Real" } EQ_Contact(in1 := "S0921_ManipulacaoReceitas_DB".RecipeEdit.C2ProfileDry.arCoffeeTemperature[9], in2 := 0.0)
      wire#w1
      { S7_Templates := "SrcType := Real" } NE_Contact(in1 := "S0921_ManipulacaoReceitas_DB".RecipeEdit.C2ProfileDry.arCoffeeTemperature[9], in2 := 0.0)
      wire#w2
      Coil( #ls_dwC2FaultProfile.%X9 )
   END_RUNG
   RUNG wire#powerrail
      { S7_Templates := "SrcType := Real" } EQ_Contact(in1 := "S0921_ManipulacaoReceitas_DB".RecipeEdit.C2ProfileDry.arInletTemperature[9], in2 := 0.0)
   END_RUNG wire#w1
   RUNG wire#powerrail
      { S7_Templates := "SrcType := Real" } EQ_Contact(in1 := "S0921_ManipulacaoReceitas_DB".RecipeEdit.C2ProfileDry.arBlowerSpeed[9], in2 := 0.0)
   END_RUNG wire#w1
   RUNG wire#w1
      { S7_Templates := "SrcType := Real" } NE_Contact(in1 := "S0921_ManipulacaoReceitas_DB".RecipeEdit.C2ProfileDry.arInletTemperature[9], in2 := 0.0)
   END_RUNG wire#w2
   RUNG wire#w1
      { S7_Templates := "SrcType := Real" } NE_Contact(in1 := "S0921_ManipulacaoReceitas_DB".RecipeEdit.C2ProfileDry.arBlowerSpeed[9], in2 := 0.0)
   END_RUNG wire#w2
   // the same network as SCL:
   #ls_dwC2FaultProfile.%X9 := (("S0921_ManipulacaoReceitas_DB".RecipeEdit.C2ProfileDry.arCoffeeTemperature[9] = 0.0) OR ("S0921_ManipulacaoReceitas_DB".RecipeEdit.C2ProfileDry.arInletTemperature[9] = 0.0) OR ("S0921_ManipulacaoReceitas_DB".RecipeEdit.C2ProfileDry.arBlowerSpeed[9] = 0.0)) AND (("S0921_ManipulacaoReceitas_DB".RecipeEdit.C2ProfileDry.arCoffeeTemperature[9] <> 0.0) OR ("S0921_ManipulacaoReceitas_DB".RecipeEdit.C2ProfileDry.arInletTemperature[9] <> 0.0) OR ("S0921_ManipulacaoReceitas_DB".RecipeEdit.C2ProfileDry.arBlowerSpeed[9] <> 0.0));
END_REGION

REGION Network 44: Falhas de receita - Linha 1 secador / Falha Profile Camara 2 - Secador Ponto 10
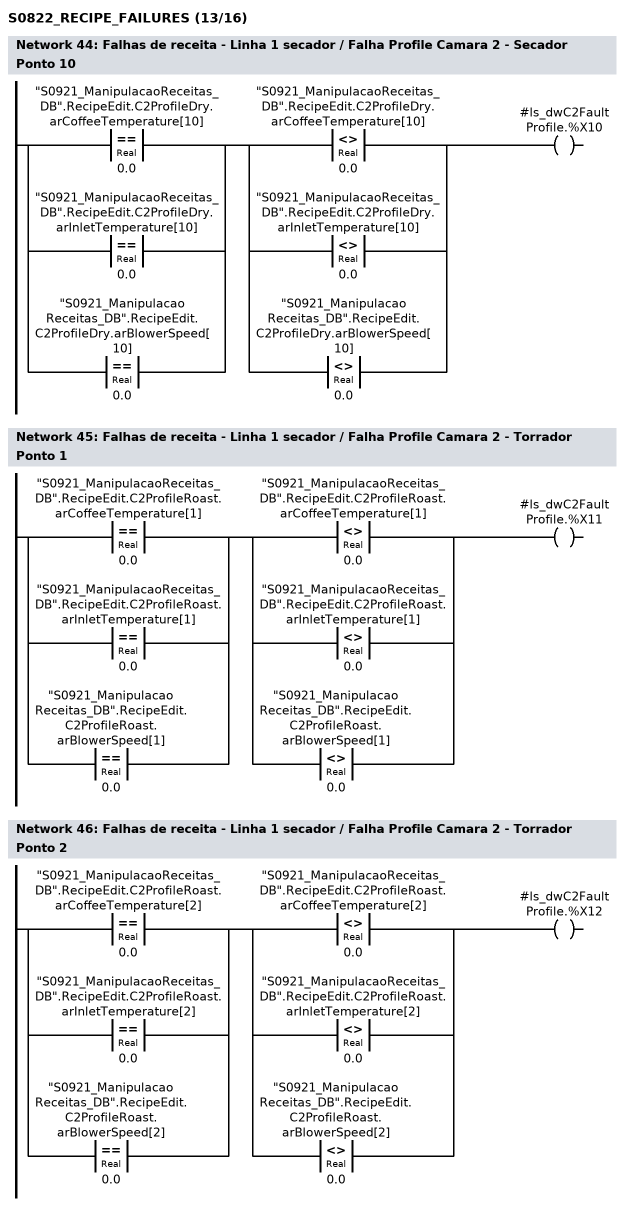
   RUNG wire#powerrail
      { S7_Templates := "SrcType := Real" } EQ_Contact(in1 := "S0921_ManipulacaoReceitas_DB".RecipeEdit.C2ProfileDry.arCoffeeTemperature[10], in2 := 0.0)
      wire#w1
      { S7_Templates := "SrcType := Real" } NE_Contact(in1 := "S0921_ManipulacaoReceitas_DB".RecipeEdit.C2ProfileDry.arCoffeeTemperature[10], in2 := 0.0)
      wire#w2
      Coil( #ls_dwC2FaultProfile.%X10 )
   END_RUNG
   RUNG wire#powerrail
      { S7_Templates := "SrcType := Real" } EQ_Contact(in1 := "S0921_ManipulacaoReceitas_DB".RecipeEdit.C2ProfileDry.arInletTemperature[10], in2 := 0.0)
   END_RUNG wire#w1
   RUNG wire#powerrail
      { S7_Templates := "SrcType := Real" } EQ_Contact(in1 := "S0921_ManipulacaoReceitas_DB".RecipeEdit.C2ProfileDry.arBlowerSpeed[10], in2 := 0.0)
   END_RUNG wire#w1
   RUNG wire#w1
      { S7_Templates := "SrcType := Real" } NE_Contact(in1 := "S0921_ManipulacaoReceitas_DB".RecipeEdit.C2ProfileDry.arInletTemperature[10], in2 := 0.0)
   END_RUNG wire#w2
   RUNG wire#w1
      { S7_Templates := "SrcType := Real" } NE_Contact(in1 := "S0921_ManipulacaoReceitas_DB".RecipeEdit.C2ProfileDry.arBlowerSpeed[10], in2 := 0.0)
   END_RUNG wire#w2
   // the same network as SCL:
   #ls_dwC2FaultProfile.%X10 := (("S0921_ManipulacaoReceitas_DB".RecipeEdit.C2ProfileDry.arCoffeeTemperature[10] = 0.0) OR ("S0921_ManipulacaoReceitas_DB".RecipeEdit.C2ProfileDry.arInletTemperature[10] = 0.0) OR ("S0921_ManipulacaoReceitas_DB".RecipeEdit.C2ProfileDry.arBlowerSpeed[10] = 0.0)) AND (("S0921_ManipulacaoReceitas_DB".RecipeEdit.C2ProfileDry.arCoffeeTemperature[10] <> 0.0) OR ("S0921_ManipulacaoReceitas_DB".RecipeEdit.C2ProfileDry.arInletTemperature[10] <> 0.0) OR ("S0921_ManipulacaoReceitas_DB".RecipeEdit.C2ProfileDry.arBlowerSpeed[10] <> 0.0));
END_REGION

REGION Network 45: Falhas de receita - Linha 1 secador / Falha Profile Camara 2 - Torrador Ponto 1
   RUNG wire#powerrail
      { S7_Templates := "SrcType := Real" } EQ_Contact(in1 := "S0921_ManipulacaoReceitas_DB".RecipeEdit.C2ProfileRoast.arCoffeeTemperature[1], in2 := 0.0)
      wire#w1
      { S7_Templates := "SrcType := Real" } NE_Contact(in1 := "S0921_ManipulacaoReceitas_DB".RecipeEdit.C2ProfileRoast.arCoffeeTemperature[1], in2 := 0.0)
      wire#w2
      Coil( #ls_dwC2FaultProfile.%X11 )
   END_RUNG
   RUNG wire#powerrail
      { S7_Templates := "SrcType := Real" } EQ_Contact(in1 := "S0921_ManipulacaoReceitas_DB".RecipeEdit.C2ProfileRoast.arInletTemperature[1], in2 := 0.0)
   END_RUNG wire#w1
   RUNG wire#powerrail
      { S7_Templates := "SrcType := Real" } EQ_Contact(in1 := "S0921_ManipulacaoReceitas_DB".RecipeEdit.C2ProfileRoast.arBlowerSpeed[1], in2 := 0.0)
   END_RUNG wire#w1
   RUNG wire#w1
      { S7_Templates := "SrcType := Real" } NE_Contact(in1 := "S0921_ManipulacaoReceitas_DB".RecipeEdit.C2ProfileRoast.arInletTemperature[1], in2 := 0.0)
   END_RUNG wire#w2
   RUNG wire#w1
      { S7_Templates := "SrcType := Real" } NE_Contact(in1 := "S0921_ManipulacaoReceitas_DB".RecipeEdit.C2ProfileRoast.arBlowerSpeed[1], in2 := 0.0)
   END_RUNG wire#w2
   // the same network as SCL:
   #ls_dwC2FaultProfile.%X11 := (("S0921_ManipulacaoReceitas_DB".RecipeEdit.C2ProfileRoast.arCoffeeTemperature[1] = 0.0) OR ("S0921_ManipulacaoReceitas_DB".RecipeEdit.C2ProfileRoast.arInletTemperature[1] = 0.0) OR ("S0921_ManipulacaoReceitas_DB".RecipeEdit.C2ProfileRoast.arBlowerSpeed[1] = 0.0)) AND (("S0921_ManipulacaoReceitas_DB".RecipeEdit.C2ProfileRoast.arCoffeeTemperature[1] <> 0.0) OR ("S0921_ManipulacaoReceitas_DB".RecipeEdit.C2ProfileRoast.arInletTemperature[1] <> 0.0) OR ("S0921_ManipulacaoReceitas_DB".RecipeEdit.C2ProfileRoast.arBlowerSpeed[1] <> 0.0));
END_REGION

REGION Network 46: Falhas de receita - Linha 1 secador / Falha Profile Camara 2 - Torrador Ponto 2
   RUNG wire#powerrail
      { S7_Templates := "SrcType := Real" } EQ_Contact(in1 := "S0921_ManipulacaoReceitas_DB".RecipeEdit.C2ProfileRoast.arCoffeeTemperature[2], in2 := 0.0)
      wire#w1
      { S7_Templates := "SrcType := Real" } NE_Contact(in1 := "S0921_ManipulacaoReceitas_DB".RecipeEdit.C2ProfileRoast.arCoffeeTemperature[2], in2 := 0.0)
      wire#w2
      Coil( #ls_dwC2FaultProfile.%X12 )
   END_RUNG
   RUNG wire#powerrail
      { S7_Templates := "SrcType := Real" } EQ_Contact(in1 := "S0921_ManipulacaoReceitas_DB".RecipeEdit.C2ProfileRoast.arInletTemperature[2], in2 := 0.0)
   END_RUNG wire#w1
   RUNG wire#powerrail
      { S7_Templates := "SrcType := Real" } EQ_Contact(in1 := "S0921_ManipulacaoReceitas_DB".RecipeEdit.C2ProfileRoast.arBlowerSpeed[2], in2 := 0.0)
   END_RUNG wire#w1
   RUNG wire#w1
      { S7_Templates := "SrcType := Real" } NE_Contact(in1 := "S0921_ManipulacaoReceitas_DB".RecipeEdit.C2ProfileRoast.arInletTemperature[2], in2 := 0.0)
   END_RUNG wire#w2
   RUNG wire#w1
      { S7_Templates := "SrcType := Real" } NE_Contact(in1 := "S0921_ManipulacaoReceitas_DB".RecipeEdit.C2ProfileRoast.arBlowerSpeed[2], in2 := 0.0)
   END_RUNG wire#w2
   // the same network as SCL:
   #ls_dwC2FaultProfile.%X12 := (("S0921_ManipulacaoReceitas_DB".RecipeEdit.C2ProfileRoast.arCoffeeTemperature[2] = 0.0) OR ("S0921_ManipulacaoReceitas_DB".RecipeEdit.C2ProfileRoast.arInletTemperature[2] = 0.0) OR ("S0921_ManipulacaoReceitas_DB".RecipeEdit.C2ProfileRoast.arBlowerSpeed[2] = 0.0)) AND (("S0921_ManipulacaoReceitas_DB".RecipeEdit.C2ProfileRoast.arCoffeeTemperature[2] <> 0.0) OR ("S0921_ManipulacaoReceitas_DB".RecipeEdit.C2ProfileRoast.arInletTemperature[2] <> 0.0) OR ("S0921_ManipulacaoReceitas_DB".RecipeEdit.C2ProfileRoast.arBlowerSpeed[2] <> 0.0));
END_REGION

REGION Network 47: Falhas de receita - Linha 1 secador / Falha Profile Camara 2 - Torrador Ponto 3
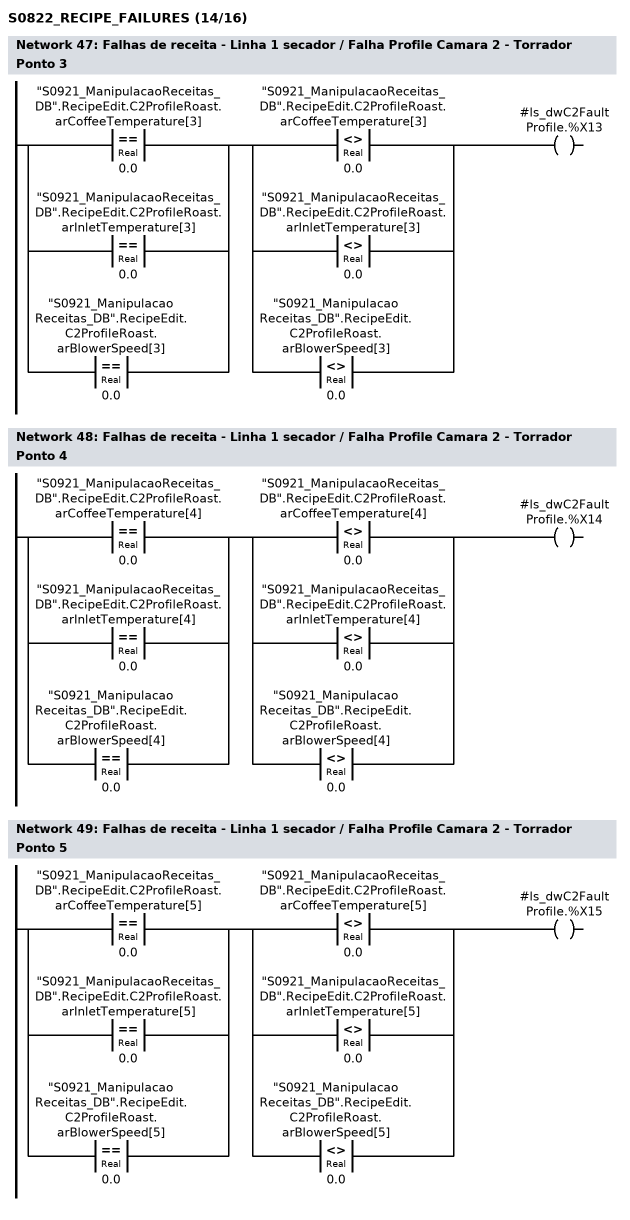
   RUNG wire#powerrail
      { S7_Templates := "SrcType := Real" } EQ_Contact(in1 := "S0921_ManipulacaoReceitas_DB".RecipeEdit.C2ProfileRoast.arCoffeeTemperature[3], in2 := 0.0)
      wire#w1
      { S7_Templates := "SrcType := Real" } NE_Contact(in1 := "S0921_ManipulacaoReceitas_DB".RecipeEdit.C2ProfileRoast.arCoffeeTemperature[3], in2 := 0.0)
      wire#w2
      Coil( #ls_dwC2FaultProfile.%X13 )
   END_RUNG
   RUNG wire#powerrail
      { S7_Templates := "SrcType := Real" } EQ_Contact(in1 := "S0921_ManipulacaoReceitas_DB".RecipeEdit.C2ProfileRoast.arInletTemperature[3], in2 := 0.0)
   END_RUNG wire#w1
   RUNG wire#powerrail
      { S7_Templates := "SrcType := Real" } EQ_Contact(in1 := "S0921_ManipulacaoReceitas_DB".RecipeEdit.C2ProfileRoast.arBlowerSpeed[3], in2 := 0.0)
   END_RUNG wire#w1
   RUNG wire#w1
      { S7_Templates := "SrcType := Real" } NE_Contact(in1 := "S0921_ManipulacaoReceitas_DB".RecipeEdit.C2ProfileRoast.arInletTemperature[3], in2 := 0.0)
   END_RUNG wire#w2
   RUNG wire#w1
      { S7_Templates := "SrcType := Real" } NE_Contact(in1 := "S0921_ManipulacaoReceitas_DB".RecipeEdit.C2ProfileRoast.arBlowerSpeed[3], in2 := 0.0)
   END_RUNG wire#w2
   // the same network as SCL:
   #ls_dwC2FaultProfile.%X13 := (("S0921_ManipulacaoReceitas_DB".RecipeEdit.C2ProfileRoast.arCoffeeTemperature[3] = 0.0) OR ("S0921_ManipulacaoReceitas_DB".RecipeEdit.C2ProfileRoast.arInletTemperature[3] = 0.0) OR ("S0921_ManipulacaoReceitas_DB".RecipeEdit.C2ProfileRoast.arBlowerSpeed[3] = 0.0)) AND (("S0921_ManipulacaoReceitas_DB".RecipeEdit.C2ProfileRoast.arCoffeeTemperature[3] <> 0.0) OR ("S0921_ManipulacaoReceitas_DB".RecipeEdit.C2ProfileRoast.arInletTemperature[3] <> 0.0) OR ("S0921_ManipulacaoReceitas_DB".RecipeEdit.C2ProfileRoast.arBlowerSpeed[3] <> 0.0));
END_REGION

REGION Network 48: Falhas de receita - Linha 1 secador / Falha Profile Camara 2 - Torrador Ponto 4
   RUNG wire#powerrail
      { S7_Templates := "SrcType := Real" } EQ_Contact(in1 := "S0921_ManipulacaoReceitas_DB".RecipeEdit.C2ProfileRoast.arCoffeeTemperature[4], in2 := 0.0)
      wire#w1
      { S7_Templates := "SrcType := Real" } NE_Contact(in1 := "S0921_ManipulacaoReceitas_DB".RecipeEdit.C2ProfileRoast.arCoffeeTemperature[4], in2 := 0.0)
      wire#w2
      Coil( #ls_dwC2FaultProfile.%X14 )
   END_RUNG
   RUNG wire#powerrail
      { S7_Templates := "SrcType := Real" } EQ_Contact(in1 := "S0921_ManipulacaoReceitas_DB".RecipeEdit.C2ProfileRoast.arInletTemperature[4], in2 := 0.0)
   END_RUNG wire#w1
   RUNG wire#powerrail
      { S7_Templates := "SrcType := Real" } EQ_Contact(in1 := "S0921_ManipulacaoReceitas_DB".RecipeEdit.C2ProfileRoast.arBlowerSpeed[4], in2 := 0.0)
   END_RUNG wire#w1
   RUNG wire#w1
      { S7_Templates := "SrcType := Real" } NE_Contact(in1 := "S0921_ManipulacaoReceitas_DB".RecipeEdit.C2ProfileRoast.arInletTemperature[4], in2 := 0.0)
   END_RUNG wire#w2
   RUNG wire#w1
      { S7_Templates := "SrcType := Real" } NE_Contact(in1 := "S0921_ManipulacaoReceitas_DB".RecipeEdit.C2ProfileRoast.arBlowerSpeed[4], in2 := 0.0)
   END_RUNG wire#w2
   // the same network as SCL:
   #ls_dwC2FaultProfile.%X14 := (("S0921_ManipulacaoReceitas_DB".RecipeEdit.C2ProfileRoast.arCoffeeTemperature[4] = 0.0) OR ("S0921_ManipulacaoReceitas_DB".RecipeEdit.C2ProfileRoast.arInletTemperature[4] = 0.0) OR ("S0921_ManipulacaoReceitas_DB".RecipeEdit.C2ProfileRoast.arBlowerSpeed[4] = 0.0)) AND (("S0921_ManipulacaoReceitas_DB".RecipeEdit.C2ProfileRoast.arCoffeeTemperature[4] <> 0.0) OR ("S0921_ManipulacaoReceitas_DB".RecipeEdit.C2ProfileRoast.arInletTemperature[4] <> 0.0) OR ("S0921_ManipulacaoReceitas_DB".RecipeEdit.C2ProfileRoast.arBlowerSpeed[4] <> 0.0));
END_REGION

REGION Network 49: Falhas de receita - Linha 1 secador / Falha Profile Camara 2 - Torrador Ponto 5
   RUNG wire#powerrail
      { S7_Templates := "SrcType := Real" } EQ_Contact(in1 := "S0921_ManipulacaoReceitas_DB".RecipeEdit.C2ProfileRoast.arCoffeeTemperature[5], in2 := 0.0)
      wire#w1
      { S7_Templates := "SrcType := Real" } NE_Contact(in1 := "S0921_ManipulacaoReceitas_DB".RecipeEdit.C2ProfileRoast.arCoffeeTemperature[5], in2 := 0.0)
      wire#w2
      Coil( #ls_dwC2FaultProfile.%X15 )
   END_RUNG
   RUNG wire#powerrail
      { S7_Templates := "SrcType := Real" } EQ_Contact(in1 := "S0921_ManipulacaoReceitas_DB".RecipeEdit.C2ProfileRoast.arInletTemperature[5], in2 := 0.0)
   END_RUNG wire#w1
   RUNG wire#powerrail
      { S7_Templates := "SrcType := Real" } EQ_Contact(in1 := "S0921_ManipulacaoReceitas_DB".RecipeEdit.C2ProfileRoast.arBlowerSpeed[5], in2 := 0.0)
   END_RUNG wire#w1
   RUNG wire#w1
      { S7_Templates := "SrcType := Real" } NE_Contact(in1 := "S0921_ManipulacaoReceitas_DB".RecipeEdit.C2ProfileRoast.arInletTemperature[5], in2 := 0.0)
   END_RUNG wire#w2
   RUNG wire#w1
      { S7_Templates := "SrcType := Real" } NE_Contact(in1 := "S0921_ManipulacaoReceitas_DB".RecipeEdit.C2ProfileRoast.arBlowerSpeed[5], in2 := 0.0)
   END_RUNG wire#w2
   // the same network as SCL:
   #ls_dwC2FaultProfile.%X15 := (("S0921_ManipulacaoReceitas_DB".RecipeEdit.C2ProfileRoast.arCoffeeTemperature[5] = 0.0) OR ("S0921_ManipulacaoReceitas_DB".RecipeEdit.C2ProfileRoast.arInletTemperature[5] = 0.0) OR ("S0921_ManipulacaoReceitas_DB".RecipeEdit.C2ProfileRoast.arBlowerSpeed[5] = 0.0)) AND (("S0921_ManipulacaoReceitas_DB".RecipeEdit.C2ProfileRoast.arCoffeeTemperature[5] <> 0.0) OR ("S0921_ManipulacaoReceitas_DB".RecipeEdit.C2ProfileRoast.arInletTemperature[5] <> 0.0) OR ("S0921_ManipulacaoReceitas_DB".RecipeEdit.C2ProfileRoast.arBlowerSpeed[5] <> 0.0));
END_REGION

REGION Network 50: Falhas de receita - Linha 1 secador / Falha Profile Camara 2 - Torrador Ponto 6
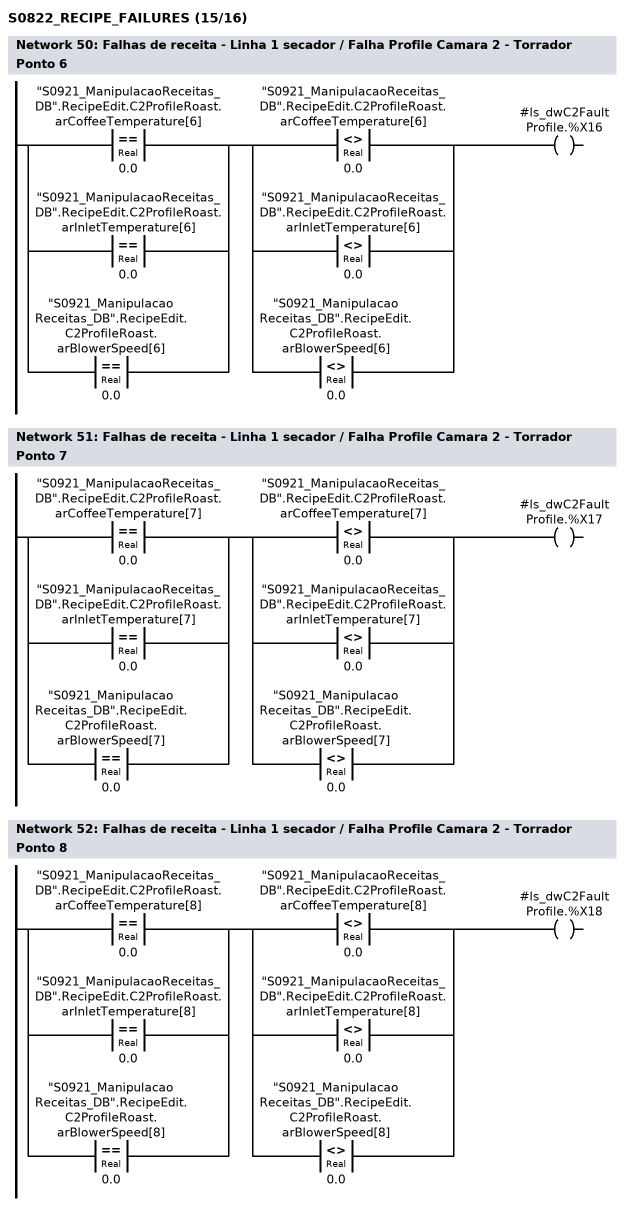
   RUNG wire#powerrail
      { S7_Templates := "SrcType := Real" } EQ_Contact(in1 := "S0921_ManipulacaoReceitas_DB".RecipeEdit.C2ProfileRoast.arCoffeeTemperature[6], in2 := 0.0)
      wire#w1
      { S7_Templates := "SrcType := Real" } NE_Contact(in1 := "S0921_ManipulacaoReceitas_DB".RecipeEdit.C2ProfileRoast.arCoffeeTemperature[6], in2 := 0.0)
      wire#w2
      Coil( #ls_dwC2FaultProfile.%X16 )
   END_RUNG
   RUNG wire#powerrail
      { S7_Templates := "SrcType := Real" } EQ_Contact(in1 := "S0921_ManipulacaoReceitas_DB".RecipeEdit.C2ProfileRoast.arInletTemperature[6], in2 := 0.0)
   END_RUNG wire#w1
   RUNG wire#powerrail
      { S7_Templates := "SrcType := Real" } EQ_Contact(in1 := "S0921_ManipulacaoReceitas_DB".RecipeEdit.C2ProfileRoast.arBlowerSpeed[6], in2 := 0.0)
   END_RUNG wire#w1
   RUNG wire#w1
      { S7_Templates := "SrcType := Real" } NE_Contact(in1 := "S0921_ManipulacaoReceitas_DB".RecipeEdit.C2ProfileRoast.arInletTemperature[6], in2 := 0.0)
   END_RUNG wire#w2
   RUNG wire#w1
      { S7_Templates := "SrcType := Real" } NE_Contact(in1 := "S0921_ManipulacaoReceitas_DB".RecipeEdit.C2ProfileRoast.arBlowerSpeed[6], in2 := 0.0)
   END_RUNG wire#w2
   // the same network as SCL:
   #ls_dwC2FaultProfile.%X16 := (("S0921_ManipulacaoReceitas_DB".RecipeEdit.C2ProfileRoast.arCoffeeTemperature[6] = 0.0) OR ("S0921_ManipulacaoReceitas_DB".RecipeEdit.C2ProfileRoast.arInletTemperature[6] = 0.0) OR ("S0921_ManipulacaoReceitas_DB".RecipeEdit.C2ProfileRoast.arBlowerSpeed[6] = 0.0)) AND (("S0921_ManipulacaoReceitas_DB".RecipeEdit.C2ProfileRoast.arCoffeeTemperature[6] <> 0.0) OR ("S0921_ManipulacaoReceitas_DB".RecipeEdit.C2ProfileRoast.arInletTemperature[6] <> 0.0) OR ("S0921_ManipulacaoReceitas_DB".RecipeEdit.C2ProfileRoast.arBlowerSpeed[6] <> 0.0));
END_REGION

REGION Network 51: Falhas de receita - Linha 1 secador / Falha Profile Camara 2 - Torrador Ponto 7
   RUNG wire#powerrail
      { S7_Templates := "SrcType := Real" } EQ_Contact(in1 := "S0921_ManipulacaoReceitas_DB".RecipeEdit.C2ProfileRoast.arCoffeeTemperature[7], in2 := 0.0)
      wire#w1
      { S7_Templates := "SrcType := Real" } NE_Contact(in1 := "S0921_ManipulacaoReceitas_DB".RecipeEdit.C2ProfileRoast.arCoffeeTemperature[7], in2 := 0.0)
      wire#w2
      Coil( #ls_dwC2FaultProfile.%X17 )
   END_RUNG
   RUNG wire#powerrail
      { S7_Templates := "SrcType := Real" } EQ_Contact(in1 := "S0921_ManipulacaoReceitas_DB".RecipeEdit.C2ProfileRoast.arInletTemperature[7], in2 := 0.0)
   END_RUNG wire#w1
   RUNG wire#powerrail
      { S7_Templates := "SrcType := Real" } EQ_Contact(in1 := "S0921_ManipulacaoReceitas_DB".RecipeEdit.C2ProfileRoast.arBlowerSpeed[7], in2 := 0.0)
   END_RUNG wire#w1
   RUNG wire#w1
      { S7_Templates := "SrcType := Real" } NE_Contact(in1 := "S0921_ManipulacaoReceitas_DB".RecipeEdit.C2ProfileRoast.arInletTemperature[7], in2 := 0.0)
   END_RUNG wire#w2
   RUNG wire#w1
      { S7_Templates := "SrcType := Real" } NE_Contact(in1 := "S0921_ManipulacaoReceitas_DB".RecipeEdit.C2ProfileRoast.arBlowerSpeed[7], in2 := 0.0)
   END_RUNG wire#w2
   // the same network as SCL:
   #ls_dwC2FaultProfile.%X17 := (("S0921_ManipulacaoReceitas_DB".RecipeEdit.C2ProfileRoast.arCoffeeTemperature[7] = 0.0) OR ("S0921_ManipulacaoReceitas_DB".RecipeEdit.C2ProfileRoast.arInletTemperature[7] = 0.0) OR ("S0921_ManipulacaoReceitas_DB".RecipeEdit.C2ProfileRoast.arBlowerSpeed[7] = 0.0)) AND (("S0921_ManipulacaoReceitas_DB".RecipeEdit.C2ProfileRoast.arCoffeeTemperature[7] <> 0.0) OR ("S0921_ManipulacaoReceitas_DB".RecipeEdit.C2ProfileRoast.arInletTemperature[7] <> 0.0) OR ("S0921_ManipulacaoReceitas_DB".RecipeEdit.C2ProfileRoast.arBlowerSpeed[7] <> 0.0));
END_REGION

REGION Network 52: Falhas de receita - Linha 1 secador / Falha Profile Camara 2 - Torrador Ponto 8
   RUNG wire#powerrail
      { S7_Templates := "SrcType := Real" } EQ_Contact(in1 := "S0921_ManipulacaoReceitas_DB".RecipeEdit.C2ProfileRoast.arCoffeeTemperature[8], in2 := 0.0)
      wire#w1
      { S7_Templates := "SrcType := Real" } NE_Contact(in1 := "S0921_ManipulacaoReceitas_DB".RecipeEdit.C2ProfileRoast.arCoffeeTemperature[8], in2 := 0.0)
      wire#w2
      Coil( #ls_dwC2FaultProfile.%X18 )
   END_RUNG
   RUNG wire#powerrail
      { S7_Templates := "SrcType := Real" } EQ_Contact(in1 := "S0921_ManipulacaoReceitas_DB".RecipeEdit.C2ProfileRoast.arInletTemperature[8], in2 := 0.0)
   END_RUNG wire#w1
   RUNG wire#powerrail
      { S7_Templates := "SrcType := Real" } EQ_Contact(in1 := "S0921_ManipulacaoReceitas_DB".RecipeEdit.C2ProfileRoast.arBlowerSpeed[8], in2 := 0.0)
   END_RUNG wire#w1
   RUNG wire#w1
      { S7_Templates := "SrcType := Real" } NE_Contact(in1 := "S0921_ManipulacaoReceitas_DB".RecipeEdit.C2ProfileRoast.arInletTemperature[8], in2 := 0.0)
   END_RUNG wire#w2
   RUNG wire#w1
      { S7_Templates := "SrcType := Real" } NE_Contact(in1 := "S0921_ManipulacaoReceitas_DB".RecipeEdit.C2ProfileRoast.arBlowerSpeed[8], in2 := 0.0)
   END_RUNG wire#w2
   // the same network as SCL:
   #ls_dwC2FaultProfile.%X18 := (("S0921_ManipulacaoReceitas_DB".RecipeEdit.C2ProfileRoast.arCoffeeTemperature[8] = 0.0) OR ("S0921_ManipulacaoReceitas_DB".RecipeEdit.C2ProfileRoast.arInletTemperature[8] = 0.0) OR ("S0921_ManipulacaoReceitas_DB".RecipeEdit.C2ProfileRoast.arBlowerSpeed[8] = 0.0)) AND (("S0921_ManipulacaoReceitas_DB".RecipeEdit.C2ProfileRoast.arCoffeeTemperature[8] <> 0.0) OR ("S0921_ManipulacaoReceitas_DB".RecipeEdit.C2ProfileRoast.arInletTemperature[8] <> 0.0) OR ("S0921_ManipulacaoReceitas_DB".RecipeEdit.C2ProfileRoast.arBlowerSpeed[8] <> 0.0));
END_REGION

REGION Network 53: Falhas de receita - Linha 1 secador / Falha Profile Camara 2 - Torrador Ponto 9
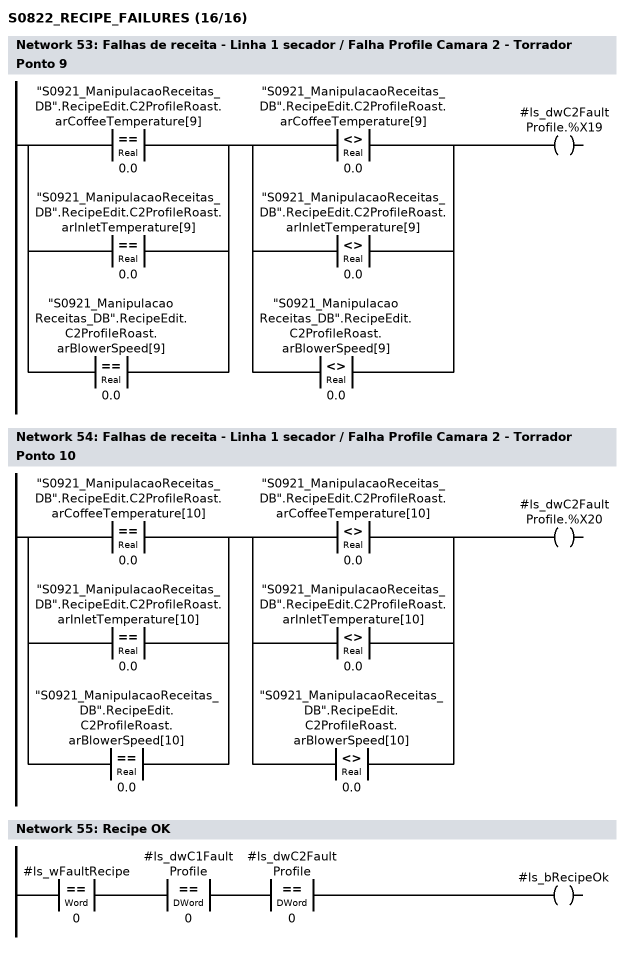
   RUNG wire#powerrail
      { S7_Templates := "SrcType := Real" } EQ_Contact(in1 := "S0921_ManipulacaoReceitas_DB".RecipeEdit.C2ProfileRoast.arCoffeeTemperature[9], in2 := 0.0)
      wire#w1
      { S7_Templates := "SrcType := Real" } NE_Contact(in1 := "S0921_ManipulacaoReceitas_DB".RecipeEdit.C2ProfileRoast.arCoffeeTemperature[9], in2 := 0.0)
      wire#w2
      Coil( #ls_dwC2FaultProfile.%X19 )
   END_RUNG
   RUNG wire#powerrail
      { S7_Templates := "SrcType := Real" } EQ_Contact(in1 := "S0921_ManipulacaoReceitas_DB".RecipeEdit.C2ProfileRoast.arInletTemperature[9], in2 := 0.0)
   END_RUNG wire#w1
   RUNG wire#powerrail
      { S7_Templates := "SrcType := Real" } EQ_Contact(in1 := "S0921_ManipulacaoReceitas_DB".RecipeEdit.C2ProfileRoast.arBlowerSpeed[9], in2 := 0.0)
   END_RUNG wire#w1
   RUNG wire#w1
      { S7_Templates := "SrcType := Real" } NE_Contact(in1 := "S0921_ManipulacaoReceitas_DB".RecipeEdit.C2ProfileRoast.arInletTemperature[9], in2 := 0.0)
   END_RUNG wire#w2
   RUNG wire#w1
      { S7_Templates := "SrcType := Real" } NE_Contact(in1 := "S0921_ManipulacaoReceitas_DB".RecipeEdit.C2ProfileRoast.arBlowerSpeed[9], in2 := 0.0)
   END_RUNG wire#w2
   // the same network as SCL:
   #ls_dwC2FaultProfile.%X19 := (("S0921_ManipulacaoReceitas_DB".RecipeEdit.C2ProfileRoast.arCoffeeTemperature[9] = 0.0) OR ("S0921_ManipulacaoReceitas_DB".RecipeEdit.C2ProfileRoast.arInletTemperature[9] = 0.0) OR ("S0921_ManipulacaoReceitas_DB".RecipeEdit.C2ProfileRoast.arBlowerSpeed[9] = 0.0)) AND (("S0921_ManipulacaoReceitas_DB".RecipeEdit.C2ProfileRoast.arCoffeeTemperature[9] <> 0.0) OR ("S0921_ManipulacaoReceitas_DB".RecipeEdit.C2ProfileRoast.arInletTemperature[9] <> 0.0) OR ("S0921_ManipulacaoReceitas_DB".RecipeEdit.C2ProfileRoast.arBlowerSpeed[9] <> 0.0));
END_REGION

REGION Network 54: Falhas de receita - Linha 1 secador / Falha Profile Camara 2 - Torrador Ponto 10
   RUNG wire#powerrail
      { S7_Templates := "SrcType := Real" } EQ_Contact(in1 := "S0921_ManipulacaoReceitas_DB".RecipeEdit.C2ProfileRoast.arCoffeeTemperature[10], in2 := 0.0)
      wire#w1
      { S7_Templates := "SrcType := Real" } NE_Contact(in1 := "S0921_ManipulacaoReceitas_DB".RecipeEdit.C2ProfileRoast.arCoffeeTemperature[10], in2 := 0.0)
      wire#w2
      Coil( #ls_dwC2FaultProfile.%X20 )
   END_RUNG
   RUNG wire#powerrail
      { S7_Templates := "SrcType := Real" } EQ_Contact(in1 := "S0921_ManipulacaoReceitas_DB".RecipeEdit.C2ProfileRoast.arInletTemperature[10], in2 := 0.0)
   END_RUNG wire#w1
   RUNG wire#powerrail
      { S7_Templates := "SrcType := Real" } EQ_Contact(in1 := "S0921_ManipulacaoReceitas_DB".RecipeEdit.C2ProfileRoast.arBlowerSpeed[10], in2 := 0.0)
   END_RUNG wire#w1
   RUNG wire#w1
      { S7_Templates := "SrcType := Real" } NE_Contact(in1 := "S0921_ManipulacaoReceitas_DB".RecipeEdit.C2ProfileRoast.arInletTemperature[10], in2 := 0.0)
   END_RUNG wire#w2
   RUNG wire#w1
      { S7_Templates := "SrcType := Real" } NE_Contact(in1 := "S0921_ManipulacaoReceitas_DB".RecipeEdit.C2ProfileRoast.arBlowerSpeed[10], in2 := 0.0)
   END_RUNG wire#w2
   // the same network as SCL:
   #ls_dwC2FaultProfile.%X20 := (("S0921_ManipulacaoReceitas_DB".RecipeEdit.C2ProfileRoast.arCoffeeTemperature[10] = 0.0) OR ("S0921_ManipulacaoReceitas_DB".RecipeEdit.C2ProfileRoast.arInletTemperature[10] = 0.0) OR ("S0921_ManipulacaoReceitas_DB".RecipeEdit.C2ProfileRoast.arBlowerSpeed[10] = 0.0)) AND (("S0921_ManipulacaoReceitas_DB".RecipeEdit.C2ProfileRoast.arCoffeeTemperature[10] <> 0.0) OR ("S0921_ManipulacaoReceitas_DB".RecipeEdit.C2ProfileRoast.arInletTemperature[10] <> 0.0) OR ("S0921_ManipulacaoReceitas_DB".RecipeEdit.C2ProfileRoast.arBlowerSpeed[10] <> 0.0));
END_REGION

REGION Network 55: Recipe OK
   RUNG wire#powerrail
      { S7_Templates := "SrcType := Word" } EQ_Contact(in1 := #ls_wFaultRecipe, in2 := 0)
      { S7_Templates := "SrcType := DWord" } EQ_Contact(in1 := #ls_dwC1FaultProfile, in2 := 0)
      { S7_Templates := "SrcType := DWord" } EQ_Contact(in1 := #ls_dwC2FaultProfile, in2 := 0)
      Coil( #ls_bRecipeOk )
   END_RUNG
   // the same network as SCL:
   #ls_bRecipeOk := (#ls_wFaultRecipe = 0) AND (#ls_dwC1FaultProfile = 0) AND (#ls_dwC2FaultProfile = 0);
END_REGION
END_FUNCTION_BLOCK
